LIN {X 0,Y 234.422,Z 1241.034,A -85,B 0,C 180,E1 12160.817,E2 12160.817} C_VEL
LIN {X 0,Y 234.7,Z 1243.569,A -85,B 0,C 180,E1 12156.114,E2 12156.114} C_VEL
LIN {X 0,Y 234.933,Z 1244.858,A -85,B 0,C 180,E1 12151.951,E2 12151.951} C_VEL
LIN {X 0,Y 234.862,Z 1245.105,A -85,B 0,C 180,E1 12147.56,E2 12147.56} C_VEL
LIN {X 0,Y 234.495,Z 1244.211,A -85,B 0,C 180,E1 12143.143,E2 12143.143} C_VEL
LIN {X 0,Y 234.238,Z 1241.662,A -85,B 0,C 180,E1 12137.833,E2 12137.833} C_VEL
LIN {X 0,Y 234.641,Z 1237.828,A -85,B 0,C 180,E1 12132.645,E2 12132.645} C_VEL
LIN {X 0,Y 235.984,Z 1232.823,A -85,B 0,C 180,E1 12127.584,E2 12127.584} C_VEL
LIN {X 0,Y 238.388,Z 1226.853,A -85,B 0,C 180,E1 12122.775,E2 12122.775} C_VEL
LIN {X 0,Y 241.931,Z 1219.741,A -85,B 0,C 180,E1 12118.061,E2 12118.061} C_VEL
LIN {X 0,Y 246.951,Z 1211.097,A -85,B 0,C 180,E1 12113.292,E2 12113.292} C_VEL
LIN {X 0,Y 255.037,Z 1198.442,A -85,B 0,C 180,E1 12107.598,E2 12107.598} C_VEL
LIN {X 0,Y 263.314,Z 1186.109,A -85,B 0,C 180,E1 12103.119,E2 12103.119} C_VEL
LIN {X 0,Y 271.68,Z 1173.895,A -85,B 0,C 180,E1 12099.387,E2 12099.387} C_VEL
LIN {X 0,Y 281.892,Z 1159.042,A -85,B 0,C 180,E1 12095.572,E2 12095.572} C_VEL
LIN {X 0,Y 294.354,Z 1140.405,A -85,B 0,C 180,E1 12091.689,E2 12091.689} C_VEL
LIN {X 0,Y 304.874,Z 1124.088,A -85,B 0,C 180,E1 12088.877,E2 12088.877} C_VEL
LIN {X 0,Y 315.79,Z 1106.483,A -85,B 0,C 180,E1 12086.314,E2 12086.314} C_VEL
LIN {X 0,Y 329.357,Z 1083.216,A -85,B 0,C 180,E1 12083.534,E2 12083.534} C_VEL
LIN {X 0,Y 339.871,Z 1063.804,A -85,B 0,C 180,E1 12081.62,E2 12081.62} C_VEL
LIN {X 0,Y 350.253,Z 1043.318,A -85,B 0,C 180,E1 12079.913,E2 12079.913} C_VEL
LIN {X 0,Y 362.426,Z 1017.02,A -85,B 0,C 180,E1 12078.118,E2 12078.118} C_VEL
LIN {X 0,Y 371.635,Z 994.992,A -85,B 0,C 180,E1 12076.892,E2 12076.892} C_VEL
LIN {X 0,Y 380.378,Z 971.962,A -85,B 0,C 180,E1 12075.829,E2 12075.829} C_VEL
LIN {X 0,Y 389.853,Z 943.44,A -85,B 0,C 180,E1 12074.781,E2 12074.781} C_VEL
LIN {X 0,Y 396.646,Z 919.703,A -85,B 0,C 180,E1 12074.096,E2 12074.096} C_VEL
LIN {X 0,Y 403.05,Z 892.634,A -85,B 0,C 180,E1 12073.424,E2 12073.424} C_VEL
LIN {X 0,Y 408.019,Z 864.078,A -85,B 0,C 180,E1 12072.829,E2 12072.829} C_VEL
LIN {X 0,Y 438.374,Z 631.58,A -85,B 0,C 180,E1 12068.871,E2 12068.871} C_VEL
LIN {X 0,Y 430.511,Z 617.928,A -85,B 0,C 180,E1 12065.23,E2 12065.23} C_VEL
LIN {X 0,Y 424.425,Z 607.912,A -85,B 0,C 180,E1 12062.059,E2 12062.059} C_VEL
LIN {X 0,Y 419.752,Z 600.312,A -85,B 0,C 180,E1 12059.318,E2 12059.318} C_VEL
LIN {X 0,Y 414.682,Z 592.173,A -85,B 0,C 180,E1 12055.99,E2 12055.99} C_VEL
LIN {X 0,Y 409.745,Z 584.609,A -85,B 0,C 180,E1 12052.287,E2 12052.287} C_VEL
LIN {X 0,Y 405.001,Z 577.41,A -85,B 0,C 180,E1 12048.031,E2 12048.031} C_VEL
LIN {X 0,Y 401.994,Z 572.607,A -85,B 0,C 180,E1 12044.713,E2 12044.713} C_VEL
LIN {X 0,Y 399.497,Z 568.951,A -85,B 0,C 180,E1 12041.466,E2 12041.466} C_VEL
LIN {X 0,Y 396.651,Z 566.18,A -85,B 0,C 180,E1 12036.939,E2 12036.939} C_VEL
LIN {X 0,Y 395.172,Z 563.252,A -85,B 0,C 180,E1 12033.274,E2 12033.274} C_VEL
LIN {X 0,Y 393.773,Z 562.552,A -85,B 0,C 180,E1 12028.839,E2 12028.839} C_VEL
LIN {X 0,Y 393.434,Z 562.231,A -85,B 0,C 180,E1 12024.165,E2 12024.165} C_VEL
LIN {X 0,Y 393.968,Z 562.553,A -85,B 0,C 180,E1 12019.363,E2 12019.363} C_VEL
LIN {X 0,Y 395.759,Z 563.395,A -85,B 0,C 180,E1 12014.617,E2 12014.617} C_VEL
LIN {X 0,Y 397.872,Z 567.235,A -85,B 0,C 180,E1 12010.183,E2 12010.183} C_VEL
LIN {X 0,Y 400.684,Z 569.721,A -85,B 0,C 180,E1 12006.53,E2 12006.53} C_VEL
LIN {X 0,Y 403.712,Z 573.853,A -85,B 0,C 180,E1 12003.16,E2 12003.16} C_VEL
LIN {X 0,Y 405.461,Z 575.63,A -85,B 0,C 180,E1 12001.603,E2 12001.603} C_VEL
LIN {X 0,Y 409.899,Z 581.322,A -85,B 0,C 180,E1 11997.927,E2 11997.927} C_VEL
LIN {X 0,Y 414.198,Z 586.829,A -85,B 0,C 180,E1 11994.906,E2 11994.906} C_VEL
LIN {X 0,Y 418.573,Z 592.702,A -85,B 0,C 180,E1 11992.174,E2 11992.174} C_VEL
LIN {X 0,Y 423.93,Z 599.787,A -85,B 0,C 180,E1 11989.245,E2 11989.245} C_VEL
LIN {X 0,Y 431.223,Z 610.33,A -85,B 0,C 180,E1 11985.706,E2 11985.706} C_VEL
LIN {X 0,Y 434.102,Z 614.761,A -85,B 0,C 180,E1 11984.42,E2 11984.42} C_VEL
LIN {X 0,Y 410.189,Z 798.407,A -85,B 0,C 180,E1 11981.329,E2 11981.329} C_VEL
LIN {X 0,Y 404.726,Z 829.257,A -85,B 0,C 180,E1 11980.609,E2 11980.609} C_VEL
LIN {X 0,Y 399.267,Z 853.642,A -85,B 0,C 180,E1 11979.878,E2 11979.878} C_VEL
LIN {X 0,Y 392.019,Z 880.927,A -85,B 0,C 180,E1 11978.876,E2 11978.876} C_VEL
LIN {X 0,Y 383.756,Z 906.782,A -85,B 0,C 180,E1 11977.701,E2 11977.701} C_VEL
LIN {X 0,Y 375.923,Z 928.552,A -85,B 0,C 180,E1 11976.525,E2 11976.525} C_VEL
LIN {X 0,Y 365.908,Z 953.393,A -85,B 0,C 180,E1 11974.938,E2 11974.938} C_VEL
LIN {X 0,Y 355.708,Z 975.722,A -85,B 0,C 180,E1 11973.223,E2 11973.223} C_VEL
LIN {X 0,Y 346.424,Z 994.396,A -85,B 0,C 180,E1 11971.551,E2 11971.551} C_VEL
LIN {X 0,Y 334.99,Z 1015.745,A -85,B 0,C 180,E1 11969.307,E2 11969.307} C_VEL
LIN {X 0,Y 323.122,Z 1035.835,A -85,B 0,C 180,E1 11966.747,E2 11966.747} C_VEL
LIN {X 0,Y 313.441,Z 1051.217,A -85,B 0,C 180,E1 11964.442,E2 11964.442} C_VEL
LIN {X 0,Y 303.132,Z 1066.743,A -85,B 0,C 180,E1 11961.716,E2 11961.716} C_VEL
LIN {X 0,Y 290.893,Z 1084.278,A -85,B 0,C 180,E1 11958.024,E2 11958.024} C_VEL
LIN {X 0,Y 280.853,Z 1097.923,A -85,B 0,C 180,E1 11954.514,E2 11954.514} C_VEL
LIN {X 0,Y 272.294,Z 1109.294,A -85,B 0,C 180,E1 11951.057,E2 11951.057} C_VEL
LIN {X 0,Y 264.585,Z 1119.425,A -85,B 0,C 180,E1 11947.433,E2 11947.433} C_VEL
LIN {X 0,Y 257.304,Z 1129.055,A -85,B 0,C 180,E1 11943.354,E2 11943.354} C_VEL
LIN {X 0,Y 249.783,Z 1139.381,A -85,B 0,C 180,E1 11938.065,E2 11938.065} C_VEL
LIN {X 0,Y 243.962,Z 1147.695,A -85,B 0,C 180,E1 11932.658,E2 11932.658} C_VEL
LIN {X 0,Y 240.175,Z 1153.774,A -85,B 0,C 180,E1 11927.821,E2 11927.821} C_VEL
LIN {X 0,Y 237.555,Z 1158.78,A -85,B 0,C 180,E1 11922.915,E2 11922.915} C_VEL
LIN {X 0,Y 235.895,Z 1162.839,A -85,B 0,C 180,E1 11917.924,E2 11917.924} C_VEL
LIN {X 0,Y 235.088,Z 1166.152,A -85,B 0,C 180,E1 11912.634,E2 11912.634} C_VEL
LIN {X 0,Y 234.883,Z 1168.717,A -85,B 0,C 180,E1 11906.823,E2 11906.823} C_VEL
LIN {X 0,Y 235.264,Z 1170.099,A -85,B 0,C 180,E1 11901.178,E2 11901.178} C_VEL
LIN {X 0,Y 236.121,Z 1170.572,A -85,B 0,C 180,E1 11895.977,E2 11895.977} C_VEL
LIN {X 0,Y 237.598,Z 1170.328,A -85,B 0,C 180,E1 11891.162,E2 11891.162} C_VEL
LIN {X 0,Y 240.343,Z 1169.243,A -85,B 0,C 180,E1 11885.97,E2 11885.97} C_VEL
LIN {X 0,Y 245.416,Z 1166.877,A -85,B 0,C 180,E1 11879.767,E2 11879.767} C_VEL
LIN {X 0,Y 253.48,Z 1162.729,A -85,B 0,C 180,E1 11873.204,E2 11873.204} C_VEL
LIN {X 0,Y 263.365,Z 1157.655,A -85,B 0,C 180,E1 11867.502,E2 11867.502} C_VEL
LIN {X 0,Y 278.43,Z 1149.865,A -85,B 0,C 180,E1 11861.143,E2 11861.143} C_VEL
LIN {X 0,Y 293.315,Z 1142.328,A -85,B 0,C 180,E1 11856.451,E2 11856.451} C_VEL
LIN {X 0,Y 295.573,Z 1141.406,A -85,B 0,C 180,E1 11855.547,E2 11855.547} C_VEL
LIN {X 0,Y 299.463,Z 1140.539,A -85,B 0,C 180,E1 11852.868,E2 11852.868} C_VEL
LIN {X 0,Y 301.764,Z 1139.659,A -85,B 0,C 180,E1 11852.154,E2 11852.154} C_VEL
LIN {X 0,Y 301.939,Z 1139.636,A -85,B 0,C 180,E1 11852.059,E2 11852.059} C_VEL
LIN {X 0,Y 275.793,Z 1163.771,A -85,B 0,C 180,E1 11845.384,E2 11845.384} C_VEL
LIN {X 0,Y 256.224,Z 1185.319,A -85,B 0,C 180,E1 11837.854,E2 11837.854} C_VEL
LIN {X 0,Y 245.979,Z 1198.298,A -85,B 0,C 180,E1 11832.284,E2 11832.284} C_VEL
LIN {X 0,Y 238.828,Z 1208.557,A -85,B 0,C 180,E1 11827.076,E2 11827.076} C_VEL
LIN {X 0,Y 233.731,Z 1217.045,A -85,B 0,C 180,E1 11822.036,E2 11822.036} C_VEL
LIN {X 0,Y 230.106,Z 1224.436,A -85,B 0,C 180,E1 11816.866,E2 11816.866} C_VEL
LIN {X 0,Y 227.883,Z 1230.405,A -85,B 0,C 180,E1 11811.898,E2 11811.898} C_VEL
LIN {X 0,Y 226.73,Z 1235.549,A -85,B 0,C 180,E1 11806.657,E2 11806.657} C_VEL
LIN {X 0,Y 226.486,Z 1239.507,A -85,B 0,C 180,E1 11801.452,E2 11801.452} C_VEL
LIN {X 0,Y 226.746,Z 1242.103,A -85,B 0,C 180,E1 11796.583,E2 11796.583} C_VEL
LIN {X 0,Y 227.037,Z 1243.443,A -85,B 0,C 180,E1 11792.271,E2 11792.271} C_VEL
LIN {X 0,Y 226.992,Z 1243.728,A -85,B 0,C 180,E1 11787.728,E2 11787.728} C_VEL
LIN {X 0,Y 226.604,Z 1242.842,A -85,B 0,C 180,E1 11783.128,E2 11783.128} C_VEL
LIN {X 0,Y 226.332,Z 1240.38,A -85,B 0,C 180,E1 11777.757,E2 11777.757} C_VEL
LIN {X 0,Y 226.769,Z 1236.476,A -85,B 0,C 180,E1 11772.288,E2 11772.288} C_VEL
LIN {X 0,Y 228.112,Z 1231.74,A -85,B 0,C 180,E1 11767.311,E2 11767.311} C_VEL
LIN {X 0,Y 230.597,Z 1225.838,A -85,B 0,C 180,E1 11762.357,E2 11762.357} C_VEL
LIN {X 0,Y 234.075,Z 1219.147,A -85,B 0,C 180,E1 11757.727,E2 11757.727} C_VEL
LIN {X 0,Y 238.931,Z 1211.085,A -85,B 0,C 180,E1 11753.064,E2 11753.064} C_VEL
LIN {X 0,Y 245.664,Z 1200.834,A -85,B 0,C 180,E1 11748.126,E2 11748.126} C_VEL
LIN {X 0,Y 255.633,Z 1186.526,A -85,B 0,C 180,E1 11742.585,E2 11742.585} C_VEL
LIN {X 0,Y 264.682,Z 1173.72,A -85,B 0,C 180,E1 11738.558,E2 11738.558} C_VEL
LIN {X 0,Y 273.854,Z 1160.76,A -85,B 0,C 180,E1 11735.13,E2 11735.13} C_VEL
LIN {X 0,Y 286.053,Z 1143.32,A -85,B 0,C 180,E1 11731.281,E2 11731.281} C_VEL
LIN {X 0,Y 298.71,Z 1124.262,A -85,B 0,C 180,E1 11727.909,E2 11727.909} C_VEL
LIN {X 0,Y 309.201,Z 1107.816,A -85,B 0,C 180,E1 11725.474,E2 11725.474} C_VEL
LIN {X 0,Y 321.711,Z 1087.238,A -85,B 0,C 180,E1 11722.918,E2 11722.918} C_VEL
LIN {X 0,Y 334.128,Z 1065.005,A -85,B 0,C 180,E1 11720.678,E2 11720.678} C_VEL
LIN {X 0,Y 344.265,Z 1045.498,A -85,B 0,C 180,E1 11719.037,E2 11719.037} C_VEL
LIN {X 0,Y 355.267,Z 1022.699,A -85,B 0,C 180,E1 11717.428,E2 11717.428} C_VEL
LIN {X 0,Y 366.125,Z 997.612,A -85,B 0,C 180,E1 11715.992,E2 11715.992} C_VEL
LIN {X 0,Y 374.666,Z 975.771,A -85,B 0,C 180,E1 11714.967,E2 11714.967} C_VEL
LIN {X 0,Y 383.02,Z 952.046,A -85,B 0,C 180,E1 11714.051,E2 11714.051} C_VEL
LIN {X 0,Y 391.563,Z 923.901,A -85,B 0,C 180,E1 11713.195,E2 11713.195} C_VEL
LIN {X 0,Y 397.58,Z 899.939,A -85,B 0,C 180,E1 11712.594,E2 11712.594} C_VEL
LIN {X 0,Y 402.75,Z 874.159,A -85,B 0,C 180,E1 11712.021,E2 11712.021} C_VEL
LIN {X 0,Y 408.292,Z 835.423,A -85,B 0,C 180,E1 11711.309,E2 11711.309} C_VEL
LIN {X 0,Y 434.7,Z 636.533,A -85,B 0,C 180,E1 11707.966,E2 11707.966} C_VEL
LIN {X 0,Y 427.973,Z 624.737,A -85,B 0,C 180,E1 11704.758,E2 11704.758} C_VEL
LIN {X 0,Y 422.268,Z 615.214,A -85,B 0,C 180,E1 11701.727,E2 11701.727} C_VEL
LIN {X 0,Y 417.624,Z 607.612,A -85,B 0,C 180,E1 11698.971,E2 11698.971} C_VEL
LIN {X 0,Y 412.699,Z 599.634,A -85,B 0,C 180,E1 11695.693,E2 11695.693} C_VEL
LIN {X 0,Y 408.17,Z 592.622,A -85,B 0,C 180,E1 11692.257,E2 11692.257} C_VEL
LIN {X 0,Y 403.583,Z 585.486,A -85,B 0,C 180,E1 11688.129,E2 11688.129} C_VEL
LIN {X 0,Y 400.287,Z 580.297,A -85,B 0,C 180,E1 11684.497,E2 11684.497} C_VEL
LIN {X 0,Y 397.874,Z 576.75,A -85,B 0,C 180,E1 11681.337,E2 11681.337} C_VEL
LIN {X 0,Y 394.986,Z 573.915,A -85,B 0,C 180,E1 11676.74,E2 11676.74} C_VEL
LIN {X 0,Y 393.634,Z 571.113,A -85,B 0,C 180,E1 11673.281,E2 11673.281} C_VEL
LIN {X 0,Y 392.232,Z 570.402,A -85,B 0,C 180,E1 11668.835,E2 11668.835} C_VEL
LIN {X 0,Y 391.893,Z 570.084,A -85,B 0,C 180,E1 11664.228,E2 11664.228} C_VEL
LIN {X 0,Y 392.428,Z 570.401,A -85,B 0,C 180,E1 11659.401,E2 11659.401} C_VEL
LIN {X 0,Y 394.169,Z 571.209,A -85,B 0,C 180,E1 11654.742,E2 11654.742} C_VEL
LIN {X 0,Y 396.379,Z 575.142,A -85,B 0,C 180,E1 11650.152,E2 11650.152} C_VEL
LIN {X 0,Y 399.044,Z 577.472,A -85,B 0,C 180,E1 11646.694,E2 11646.694} C_VEL
LIN {X 0,Y 402.228,Z 581.766,A -85,B 0,C 180,E1 11643.154,E2 11643.154} C_VEL
LIN {X 0,Y 403.777,Z 583.406,A -85,B 0,C 180,E1 11641.75,E2 11641.75} C_VEL
LIN {X 0,Y 408.145,Z 589.012,A -85,B 0,C 180,E1 11638.122,E2 11638.122} C_VEL
LIN {X 0,Y 412.383,Z 594.497,A -85,B 0,C 180,E1 11635.107,E2 11635.107} C_VEL
LIN {X 0,Y 416.581,Z 600.152,A -85,B 0,C 180,E1 11632.468,E2 11632.468} C_VEL
LIN {X 0,Y 421.918,Z 607.271,A -85,B 0,C 180,E1 11629.521,E2 11629.521} C_VEL
LIN {X 0,Y 429.179,Z 617.87,A -85,B 0,C 180,E1 11625.957,E2 11625.957} C_VEL
LIN {X 0,Y 430.532,Z 620.121,A -85,B 0,C 180,E1 11625.326,E2 11625.326} C_VEL
LIN {X 0,Y 406.793,Z 798.694,A -85,B 0,C 180,E1 11622.345,E2 11622.345} C_VEL
LIN {X 0,Y 401.234,Z 829.703,A -85,B 0,C 180,E1 11621.631,E2 11621.631} C_VEL
LIN {X 0,Y 395.799,Z 853.696,A -85,B 0,C 180,E1 11620.922,E2 11620.922} C_VEL
LIN {X 0,Y 388.651,Z 880.41,A -85,B 0,C 180,E1 11619.96,E2 11619.96} C_VEL
LIN {X 0,Y 380.1,Z 906.91,A -85,B 0,C 180,E1 11618.776,E2 11618.776} C_VEL
LIN {X 0,Y 372.259,Z 928.403,A -85,B 0,C 180,E1 11617.631,E2 11617.631} C_VEL
LIN {X 0,Y 362.311,Z 952.866,A -85,B 0,C 180,E1 11616.098,E2 11616.098} C_VEL
LIN {X 0,Y 351.313,Z 976.538,A -85,B 0,C 180,E1 11614.3,E2 11614.3} C_VEL
LIN {X 0,Y 342.082,Z 994.772,A -85,B 0,C 180,E1 11612.681,E2 11612.681} C_VEL
LIN {X 0,Y 330.982,Z 1015.11,A -85,B 0,C 180,E1 11610.567,E2 11610.567} C_VEL
LIN {X 0,Y 318.185,Z 1036.478,A -85,B 0,C 180,E1 11607.877,E2 11607.877} C_VEL
LIN {X 0,Y 307.923,Z 1052.44,A -85,B 0,C 180,E1 11605.486,E2 11605.486} C_VEL
LIN {X 0,Y 297.791,Z 1067.386,A -85,B 0,C 180,E1 11602.864,E2 11602.864} C_VEL
LIN {X 0,Y 285.709,Z 1084.402,A -85,B 0,C 180,E1 11599.311,E2 11599.311} C_VEL
LIN {X 0,Y 274.386,Z 1099.39,A -85,B 0,C 180,E1 11595.437,E2 11595.437} C_VEL
LIN {X 0,Y 265.188,Z 1111.244,A -85,B 0,C 180,E1 11591.763,E2 11591.763} C_VEL
LIN {X 0,Y 256.212,Z 1122.705,A -85,B 0,C 180,E1 11587.515,E2 11587.515} C_VEL
LIN {X 0,Y 246.831,Z 1134.724,A -85,B 0,C 180,E1 11581.972,E2 11581.972} C_VEL
LIN {X 0,Y 240.673,Z 1142.891,A -85,B 0,C 180,E1 11577.311,E2 11577.311} C_VEL
LIN {X 0,Y 235.936,Z 1149.613,A -85,B 0,C 180,E1 11572.698,E2 11572.698} C_VEL
LIN {X 0,Y 232.166,Z 1155.527,A -85,B 0,C 180,E1 11567.79,E2 11567.79} C_VEL
LIN {X 0,Y 229.434,Z 1160.696,A -85,B 0,C 180,E1 11562.493,E2 11562.493} C_VEL
LIN {X 0,Y 227.574,Z 1165.693,A -85,B 0,C 180,E1 11555.758,E2 11555.758} C_VEL
LIN {X 0,Y 227.033,Z 1168.637,A -85,B 0,C 180,E1 11550.138,E2 11550.138} C_VEL
LIN {X 0,Y 227.051,Z 1170.514,A -85,B 0,C 180,E1 11545.01,E2 11545.01} C_VEL
LIN {X 0,Y 227.501,Z 1171.634,A -85,B 0,C 180,E1 11540.049,E2 11540.049} C_VEL
LIN {X 0,Y 228.425,Z 1172.094,A -85,B 0,C 180,E1 11535.227,E2 11535.227} C_VEL
LIN {X 0,Y 230.104,Z 1171.893,A -85,B 0,C 180,E1 11530.263,E2 11530.263} C_VEL
LIN {X 0,Y 233.156,Z 1170.882,A -85,B 0,C 180,E1 11524.92,E2 11524.92} C_VEL
LIN {X 0,Y 239.244,Z 1168.447,A -85,B 0,C 180,E1 11518.084,E2 11518.084} C_VEL
LIN {X 0,Y 248.147,Z 1164.309,A -85,B 0,C 180,E1 11511.426,E2 11511.426} C_VEL
LIN {X 0,Y 260.72,Z 1158.606,A -85,B 0,C 180,E1 11504.883,E2 11504.883} C_VEL
LIN {X 0,Y 279.21,Z 1149.934,A -85,B 0,C 180,E1 11498.048,E2 11498.048} C_VEL
LIN {X 0,Y 301.113,Z 1139.941,A -85,B 0,C 180,E1 11492.297,E2 11492.297} C_VEL
LIN {X 0,Y 301.764,Z 1139.659,A -85,B 0,C 180,E1 11492.154,E2 11492.154} C_VEL
LIN {X 0,Y 302.162,Z 1139.777,A -85,B 0,C 180,E1 11491.778,E2 11491.778} C_VEL
LIN {X 0,Y 300.773,Z 1141.241,A -85,B 0,C 180,E1 11491.224,E2 11491.224} C_VEL
LIN {X 0,Y 296.315,Z 1144.749,A -85,B 0,C 180,E1 11490.576,E2 11490.576} C_VEL
LIN {X 0,Y 282.499,Z 1154.252,A -85,B 0,C 180,E1 11489.503,E2 11489.503} C_VEL
LIN {X 0,Y 278.089,Z 1157.541,A -85,B 0,C 180,E1 11488.81,E2 11488.81} C_VEL
LIN {X 0,Y 277.288,Z 1158.24,A -85,B 0,C 180,E1 11488.611,E2 11488.611} C_VEL
LIN {X 0,Y 253.039,Z 1182.018,A -85,B 0,C 180,E1 11480.402,E2 11480.402} C_VEL
LIN {X 0,Y 240.686,Z 1196.16,A -85,B 0,C 180,E1 11474.26,E2 11474.26} C_VEL
LIN {X 0,Y 232.339,Z 1207.025,A -85,B 0,C 180,E1 11468.609,E2 11468.609} C_VEL
LIN {X 0,Y 226.553,Z 1215.843,A -85,B 0,C 180,E1 11463.179,E2 11463.179} C_VEL
LIN {X 0,Y 222.525,Z 1223.309,A -85,B 0,C 180,E1 11457.724,E2 11457.724} C_VEL
LIN {X 0,Y 220.065,Z 1229.357,A -85,B 0,C 180,E1 11452.436,E2 11452.436} C_VEL
LIN {X 0,Y 218.853,Z 1234.201,A -85,B 0,C 180,E1 11447.275,E2 11447.275} C_VEL
LIN {X 0,Y 218.54,Z 1237.967,A -85,B 0,C 180,E1 11442.149,E2 11442.149} C_VEL
LIN {X 0,Y 218.771,Z 1240.528,A -85,B 0,C 180,E1 11437.342,E2 11437.342} C_VEL
LIN {X 0,Y 219.117,Z 1241.981,A -85,B 0,C 180,E1 11432.877,E2 11432.877} C_VEL
LIN {X 0,Y 219.13,Z 1242.384,A -85,B 0,C 180,E1 11428.17,E2 11428.17} C_VEL
LIN {X 0,Y 218.743,Z 1241.599,A -85,B 0,C 180,E1 11423.438,E2 11423.438} C_VEL
LIN {X 0,Y 218.426,Z 1239.193,A -85,B 0,C 180,E1 11417.844,E2 11417.844} C_VEL
LIN {X 0,Y 218.852,Z 1235.35,A -85,B 0,C 180,E1 11412.175,E2 11412.175} C_VEL
LIN {X 0,Y 220.356,Z 1230.382,A -85,B 0,C 180,E1 11406.749,E2 11406.749} C_VEL
LIN {X 0,Y 223.001,Z 1224.465,A -85,B 0,C 180,E1 11401.623,E2 11401.623} C_VEL
LIN {X 0,Y 226.702,Z 1217.743,A -85,B 0,C 180,E1 11396.845,E2 11396.845} C_VEL
LIN {X 0,Y 231.95,Z 1209.439,A -85,B 0,C 180,E1 11391.944,E2 11391.944} C_VEL
LIN {X 0,Y 240.114,Z 1197.738,A -85,B 0,C 180,E1 11386.271,E2 11386.271} C_VEL
LIN {X 0,Y 249.719,Z 1184.4,A -85,B 0,C 180,E1 11381.17,E2 11381.17} C_VEL
LIN {X 0,Y 258.803,Z 1172.049,A -85,B 0,C 180,E1 11377.262,E2 11377.262} C_VEL
LIN {X 0,Y 269.514,Z 1157.448,A -85,B 0,C 180,E1 11373.412,E2 11373.412} C_VEL
LIN {X 0,Y 282.806,Z 1138.8,A -85,B 0,C 180,E1 11369.436,E2 11369.436} C_VEL
LIN {X 0,Y 293.673,Z 1122.857,A -85,B 0,C 180,E1 11366.653,E2 11366.653} C_VEL
LIN {X 0,Y 304.682,Z 1105.965,A -85,B 0,C 180,E1 11364.173,E2 11364.173} C_VEL
LIN {X 0,Y 318.14,Z 1084.13,A -85,B 0,C 180,E1 11361.52,E2 11361.52} C_VEL
LIN {X 0,Y 330.237,Z 1062.753,A -85,B 0,C 180,E1 11359.413,E2 11359.413} C_VEL
LIN {X 0,Y 340.729,Z 1042.858,A -85,B 0,C 180,E1 11357.77,E2 11357.77} C_VEL
LIN {X 0,Y 352.76,Z 1018.101,A -85,B 0,C 180,E1 11356.081,E2 11356.081} C_VEL
LIN {X 0,Y 362.978,Z 994.576,A -85,B 0,C 180,E1 11354.787,E2 11354.787} C_VEL
LIN {X 0,Y 371.662,Z 972.557,A -85,B 0,C 180,E1 11353.786,E2 11353.786} C_VEL
LIN {X 0,Y 381.161,Z 945.476,A -85,B 0,C 180,E1 11352.79,E2 11352.79} C_VEL
LIN {X 0,Y 388.711,Z 920.179,A -85,B 0,C 180,E1 11352.07,E2 11352.07} C_VEL
LIN {X 0,Y 394.526,Z 896.939,A -85,B 0,C 180,E1 11351.499,E2 11351.499} C_VEL
LIN {X 0,Y 400.202,Z 868.074,A -85,B 0,C 180,E1 11350.876,E2 11350.876} C_VEL
LIN {X 0,Y 407.304,Z 816.655,A -85,B 0,C 180,E1 11349.97,E2 11349.97} C_VEL
LIN {X 0,Y 431.165,Z 641.595,A -85,B 0,C 180,E1 11347.06,E2 11347.06} C_VEL
LIN {X 0,Y 424.708,Z 630.234,A -85,B 0,C 180,E1 11343.881,E2 11343.881} C_VEL
LIN {X 0,Y 418.475,Z 619.575,A -85,B 0,C 180,E1 11340.411,E2 11340.411} C_VEL
LIN {X 0,Y 412.079,Z 609.24,A -85,B 0,C 180,E1 11336.313,E2 11336.313} C_VEL
LIN {X 0,Y 407.153,Z 601.482,A -85,B 0,C 180,E1 11332.663,E2 11332.663} C_VEL
LIN {X 0,Y 404.391,Z 597.255,A -85,B 0,C 180,E1 11330.32,E2 11330.32} C_VEL
LIN {X 0,Y 401.42,Z 592.59,A -85,B 0,C 180,E1 11327.484,E2 11327.484} C_VEL
LIN {X 0,Y 398.585,Z 587.986,A -85,B 0,C 180,E1 11324.28,E2 11324.28} C_VEL
LIN {X 0,Y 396.333,Z 584.602,A -85,B 0,C 180,E1 11321.313,E2 11321.313} C_VEL
LIN {X 0,Y 393.384,Z 581.722,A -85,B 0,C 180,E1 11316.639,E2 11316.639} C_VEL
LIN {X 0,Y 392.04,Z 578.925,A -85,B 0,C 180,E1 11313.164,E2 11313.164} C_VEL
LIN {X 0,Y 390.7,Z 578.255,A -85,B 0,C 180,E1 11308.871,E2 11308.871} C_VEL
LIN {X 0,Y 390.35,Z 577.935,A -85,B 0,C 180,E1 11304.265,E2 11304.265} C_VEL
LIN {X 0,Y 390.888,Z 578.249,A -85,B 0,C 180,E1 11299.439,E2 11299.439} C_VEL
LIN {X 0,Y 392.593,Z 579.04,A -85,B 0,C 180,E1 11294.821,E2 11294.821} C_VEL
LIN {X 0,Y 394.759,Z 582.904,A -85,B 0,C 180,E1 11290.323,E2 11290.323} C_VEL
LIN {X 0,Y 397.407,Z 585.224,A -85,B 0,C 180,E1 11286.86,E2 11286.86} C_VEL
LIN {X 0,Y 400.619,Z 589.562,A -85,B 0,C 180,E1 11283.267,E2 11283.267} C_VEL
LIN {X 0,Y 402.096,Z 591.18,A -85,B 0,C 180,E1 11281.898,E2 11281.898} C_VEL
LIN {X 0,Y 406.324,Z 596.624,A -85,B 0,C 180,E1 11278.355,E2 11278.355} C_VEL
LIN {X 0,Y 410.643,Z 602.266,A -85,B 0,C 180,E1 11275.263,E2 11275.263} C_VEL
LIN {X 0,Y 414.721,Z 607.772,A -85,B 0,C 180,E1 11272.691,E2 11272.691} C_VEL
LIN {X 0,Y 419.978,Z 614.868,A -85,B 0,C 180,E1 11269.759,E2 11269.759} C_VEL
LIN {X 0,Y 427.04,Z 625.276,A -85,B 0,C 180,E1 11266.248,E2 11266.248} C_VEL
LIN {X 0,Y 403.207,Z 800.417,A -85,B 0,C 180,E1 11263.343,E2 11263.343} C_VEL
LIN {X 0,Y 397.539,Z 831.173,A -85,B 0,C 180,E1 11262.636,E2 11262.636} C_VEL
LIN {X 0,Y 391.957,Z 855.307,A -85,B 0,C 180,E1 11261.925,E2 11261.925} C_VEL
LIN {X 0,Y 384.476,Z 882.596,A -85,B 0,C 180,E1 11260.944,E2 11260.944} C_VEL
LIN {X 0,Y 375.996,Z 908.327,A -85,B 0,C 180,E1 11259.799,E2 11259.799} C_VEL
LIN {X 0,Y 367.899,Z 930.148,A -85,B 0,C 180,E1 11258.644,E2 11258.644} C_VEL
LIN {X 0,Y 357.452,Z 955.255,A -85,B 0,C 180,E1 11257.07,E2 11257.07} C_VEL
LIN {X 0,Y 346.783,Z 977.834,A -85,B 0,C 180,E1 11255.362,E2 11255.362} C_VEL
LIN {X 0,Y 336.878,Z 997.036,A -85,B 0,C 180,E1 11253.659,E2 11253.659} C_VEL
LIN {X 0,Y 324.315,Z 1019.4,A -85,B 0,C 180,E1 11251.297,E2 11251.297} C_VEL
LIN {X 0,Y 312.728,Z 1038.135,A -85,B 0,C 180,E1 11248.901,E2 11248.901} C_VEL
LIN {X 0,Y 302.511,Z 1053.657,A -85,B 0,C 180,E1 11246.569,E2 11246.569} C_VEL
LIN {X 0,Y 292.022,Z 1068.759,A -85,B 0,C 180,E1 11243.907,E2 11243.907} C_VEL
LIN {X 0,Y 279.613,Z 1085.757,A -85,B 0,C 180,E1 11240.325,E2 11240.325} C_VEL
LIN {X 0,Y 268.342,Z 1100.276,A -85,B 0,C 180,E1 11236.542,E2 11236.542} C_VEL
LIN {X 0,Y 259.145,Z 1111.819,A -85,B 0,C 180,E1 11232.948,E2 11232.948} C_VEL
LIN {X 0,Y 250.579,Z 1122.413,A -85,B 0,C 180,E1 11229.025,E2 11229.025} C_VEL
LIN {X 0,Y 241.298,Z 1134.052,A -85,B 0,C 180,E1 11223.803,E2 11223.803} C_VEL
LIN {X 0,Y 233.349,Z 1144.081,A -85,B 0,C 180,E1 11218.041,E2 11218.041} C_VEL
LIN {X 0,Y 228.243,Z 1151.066,A -85,B 0,C 180,E1 11213.119,E2 11213.119} C_VEL
LIN {X 0,Y 224.164,Z 1157.28,A -85,B 0,C 180,E1 11207.77,E2 11207.77} C_VEL
LIN {X 0,Y 221.065,Z 1163.226,A -85,B 0,C 180,E1 11201.328,E2 11201.328} C_VEL
LIN {X 0,Y 219.579,Z 1167.268,A -85,B 0,C 180,E1 11195.332,E2 11195.332} C_VEL
LIN {X 0,Y 219.133,Z 1169.926,A -85,B 0,C 180,E1 11190.128,E2 11190.128} C_VEL
LIN {X 0,Y 219.168,Z 1171.888,A -85,B 0,C 180,E1 11184.788,E2 11184.788} C_VEL
LIN {X 0,Y 219.685,Z 1173.097,A -85,B 0,C 180,E1 11179.586,E2 11179.586} C_VEL
LIN {X 0,Y 220.767,Z 1173.62,A -85,B 0,C 180,E1 11174.425,E2 11174.425} C_VEL
LIN {X 0,Y 222.814,Z 1173.456,A -85,B 0,C 180,E1 11169.037,E2 11169.037} C_VEL
LIN {X 0,Y 226.363,Z 1172.464,A -85,B 0,C 180,E1 11163.37,E2 11163.37} C_VEL
LIN {X 0,Y 233.502,Z 1169.924,A -85,B 0,C 180,E1 11156.132,E2 11156.132} C_VEL
LIN {X 0,Y 243.502,Z 1165.818,A -85,B 0,C 180,E1 11149.351,E2 11149.351} C_VEL
LIN {X 0,Y 257.818,Z 1159.904,A -85,B 0,C 180,E1 11142.562,E2 11142.562} C_VEL
LIN {X 0,Y 277.458,Z 1151.727,A -85,B 0,C 180,E1 11135.969,E2 11135.969} C_VEL
LIN {X 0,Y 292.187,Z 1145.694,A -85,B 0,C 180,E1 11132.186,E2 11132.186} C_VEL
LIN {X 0,Y 277.288,Z 1158.24,A -85,B 0,C 180,E1 11128.611,E2 11128.611} C_VEL
LIN {X 0,Y 272.552,Z 1162.19,A -85,B 0,C 180,E1 11127.615,E2 11127.615} C_VEL
LIN {X 0,Y 257.615,Z 1172.667,A -85,B 0,C 180,E1 11125.281,E2 11125.281} C_VEL
LIN {X 0,Y 253.807,Z 1175.745,A -85,B 0,C 180,E1 11124.273,E2 11124.273} C_VEL
LIN {X 0,Y 236.34,Z 1193.39,A -85,B 0,C 180,E1 11116.691,E2 11116.691} C_VEL
LIN {X 0,Y 226.399,Z 1205.124,A -85,B 0,C 180,E1 11110.482,E2 11110.482} C_VEL
LIN {X 0,Y 219.21,Z 1215.079,A -85,B 0,C 180,E1 11104.127,E2 11104.127} C_VEL
LIN {X 0,Y 213.708,Z 1224.89,A -85,B 0,C 180,E1 11096.39,E2 11096.39} C_VEL
LIN {X 0,Y 211.221,Z 1231.706,A -85,B 0,C 180,E1 11089.352,E2 11089.352} C_VEL
LIN {X 0,Y 210.59,Z 1235.932,A -85,B 0,C 180,E1 11083.733,E2 11083.733} C_VEL
LIN {X 0,Y 210.761,Z 1238.824,A -85,B 0,C 180,E1 11078.457,E2 11078.457} C_VEL
LIN {X 0,Y 211.192,Z 1240.509,A -85,B 0,C 180,E1 11073.529,E2 11073.529} C_VEL
LIN {X 0,Y 211.255,Z 1241.028,A -85,B 0,C 180,E1 11068.915,E2 11068.915} C_VEL
LIN {X 0,Y 210.959,Z 1240.403,A -85,B 0,C 180,E1 11064.288,E2 11064.288} C_VEL
LIN {X 0,Y 210.533,Z 1238.308,A -85,B 0,C 180,E1 11058.494,E2 11058.494} C_VEL
LIN {X 0,Y 210.94,Z 1234.194,A -85,B 0,C 180,E1 11052.055,E2 11052.055} C_VEL
LIN {X 0,Y 212.504,Z 1229.264,A -85,B 0,C 180,E1 11046.425,E2 11046.425} C_VEL
LIN {X 0,Y 215.264,Z 1223.37,A -85,B 0,C 180,E1 11041.114,E2 11041.114} C_VEL
LIN {X 0,Y 219.177,Z 1216.606,A -85,B 0,C 180,E1 11036.129,E2 11036.129} C_VEL
LIN {X 0,Y 224.501,Z 1208.557,A -85,B 0,C 180,E1 11031.208,E2 11031.208} C_VEL
LIN {X 0,Y 231.891,Z 1198.313,A -85,B 0,C 180,E1 11026.036,E2 11026.036} C_VEL
LIN {X 0,Y 242.606,Z 1184.091,A -85,B 0,C 180,E1 11020.318,E2 11020.318} C_VEL
LIN {X 0,Y 251.957,Z 1171.823,A -85,B 0,C 180,E1 11016.332,E2 11016.332} C_VEL
LIN {X 0,Y 261.75,Z 1158.862,A -85,B 0,C 180,E1 11012.818,E2 11012.818} C_VEL
LIN {X 0,Y 273.718,Z 1142.73,A -85,B 0,C 180,E1 11009.185,E2 11009.185} C_VEL
LIN {X 0,Y 287.358,Z 1123.384,A -85,B 0,C 180,E1 11005.683,E2 11005.683} C_VEL
LIN {X 0,Y 298.587,Z 1106.638,A -85,B 0,C 180,E1 11003.188,E2 11003.188} C_VEL
LIN {X 0,Y 310.733,Z 1087.539,A -85,B 0,C 180,E1 11000.809,E2 11000.809} C_VEL
LIN {X 0,Y 324.596,Z 1063.941,A -85,B 0,C 180,E1 10998.422,E2 10998.422} C_VEL
LIN {X 0,Y 335.244,Z 1044.278,A -85,B 0,C 180,E1 10996.786,E2 10996.786} C_VEL
LIN {X 0,Y 346.182,Z 1022.497,A -85,B 0,C 180,E1 10995.271,E2 10995.271} C_VEL
LIN {X 0,Y 358.248,Z 995.74,A -85,B 0,C 180,E1 10993.767,E2 10993.767} C_VEL
LIN {X 0,Y 367.043,Z 973.97,A -85,B 0,C 180,E1 10992.777,E2 10992.777} C_VEL
LIN {X 0,Y 375.98,Z 949.329,A -85,B 0,C 180,E1 10991.86,E2 10991.86} C_VEL
LIN {X 0,Y 384.819,Z 920.801,A -85,B 0,C 180,E1 10991.036,E2 10991.036} C_VEL
LIN {X 0,Y 390.941,Z 896.874,A -85,B 0,C 180,E1 10990.454,E2 10990.454} C_VEL
LIN {X 0,Y 396.731,Z 868.302,A -85,B 0,C 180,E1 10989.84,E2 10989.84} C_VEL
LIN {X 0,Y 404.892,Z 810.837,A -85,B 0,C 180,E1 10988.835,E2 10988.835} C_VEL
LIN {X 0,Y 427.68,Z 646.546,A -85,B 0,C 180,E1 10986.128,E2 10986.128} C_VEL
LIN {X 0,Y 420.731,Z 634.384,A -85,B 0,C 180,E1 10982.588,E2 10982.588} C_VEL
LIN {X 0,Y 414.623,Z 624.067,A -85,B 0,C 180,E1 10979.033,E2 10979.033} C_VEL
LIN {X 0,Y 409.051,Z 614.975,A -85,B 0,C 180,E1 10975.303,E2 10975.303} C_VEL
LIN {X 0,Y 404.83,Z 608.356,A -85,B 0,C 180,E1 10972.05,E2 10972.05} C_VEL
LIN {X 0,Y 402.068,Z 604.104,A -85,B 0,C 180,E1 10969.613,E2 10969.613} C_VEL
LIN {X 0,Y 399.643,Z 600.178,A -85,B 0,C 180,E1 10967.207,E2 10967.207} C_VEL
LIN {X 0,Y 396.889,Z 595.675,A -85,B 0,C 180,E1 10964.061,E2 10964.061} C_VEL
LIN {X 0,Y 394.636,Z 592.347,A -85,B 0,C 180,E1 10961.076,E2 10961.076} C_VEL
LIN {X 0,Y 391.693,Z 589.409,A -85,B 0,C 180,E1 10956.373,E2 10956.373} C_VEL
LIN {X 0,Y 390.438,Z 586.73,A -85,B 0,C 180,E1 10953.024,E2 10953.024} C_VEL
LIN {X 0,Y 389.133,Z 586.094,A -85,B 0,C 180,E1 10948.732,E2 10948.732} C_VEL
LIN {X 0,Y 388.806,Z 585.773,A -85,B 0,C 180,E1 10943.919,E2 10943.919} C_VEL
LIN {X 0,Y 389.39,Z 586.124,A -85,B 0,C 180,E1 10939.244,E2 10939.244} C_VEL
LIN {X 0,Y 391.045,Z 586.99,A -85,B 0,C 180,E1 10934.801,E2 10934.801} C_VEL
LIN {X 0,Y 393.304,Z 590.859,A -85,B 0,C 180,E1 10930.22,E2 10930.22} C_VEL
LIN {X 0,Y 395.82,Z 593.076,A -85,B 0,C 180,E1 10926.956,E2 10926.956} C_VEL
LIN {X 0,Y 399.183,Z 597.517,A -85,B 0,C 180,E1 10923.215,E2 10923.215} C_VEL
LIN {X 0,Y 400.419,Z 598.953,A -85,B 0,C 180,E1 10922.048,E2 10922.048} C_VEL
LIN {X 0,Y 404.646,Z 604.441,A -85,B 0,C 180,E1 10918.483,E2 10918.483} C_VEL
LIN {X 0,Y 408.68,Z 609.703,A -85,B 0,C 180,E1 10915.576,E2 10915.576} C_VEL
LIN {X 0,Y 413.078,Z 615.685,A -85,B 0,C 180,E1 10912.786,E2 10912.786} C_VEL
LIN {X 0,Y 418.223,Z 622.795,A -85,B 0,C 180,E1 10909.882,E2 10909.882} C_VEL
LIN {X 0,Y 423.535,Z 630.753,A -85,B 0,C 180,E1 10907.175,E2 10907.175} C_VEL
LIN {X 0,Y 399.897,Z 801.083,A -85,B 0,C 180,E1 10904.378,E2 10904.378} C_VEL
LIN {X 0,Y 394.095,Z 832.069,A -85,B 0,C 180,E1 10903.674,E2 10903.674} C_VEL
LIN {X 0,Y 388.412,Z 856.192,A -85,B 0,C 180,E1 10902.97,E2 10902.97} C_VEL
LIN {X 0,Y 381.011,Z 882.822,A -85,B 0,C 180,E1 10902.026,E2 10902.026} C_VEL
LIN {X 0,Y 372.284,Z 908.942,A -85,B 0,C 180,E1 10900.881,E2 10900.881} C_VEL
LIN {X 0,Y 363.786,Z 931.451,A -85,B 0,C 180,E1 10899.702,E2 10899.702} C_VEL
LIN {X 0,Y 353.141,Z 956.526,A -85,B 0,C 180,E1 10898.139,E2 10898.139} C_VEL
LIN {X 0,Y 342.828,Z 978.001,A -85,B 0,C 180,E1 10896.531,E2 10896.531} C_VEL
LIN {X 0,Y 333.196,Z 996.409,A -85,B 0,C 180,E1 10894.926,E2 10894.926} C_VEL
LIN {X 0,Y 322.402,Z 1015.509,A -85,B 0,C 180,E1 10892.979,E2 10892.979} C_VEL
LIN {X 0,Y 308.972,Z 1037.289,A -85,B 0,C 180,E1 10890.304,E2 10890.304} C_VEL
LIN {X 0,Y 297.773,Z 1054.041,A -85,B 0,C 180,E1 10887.823,E2 10887.823} C_VEL
LIN {X 0,Y 286.993,Z 1069.252,A -85,B 0,C 180,E1 10885.161,E2 10885.161} C_VEL
LIN {X 0,Y 273.984,Z 1086.652,A -85,B 0,C 180,E1 10881.497,E2 10881.497} C_VEL
LIN {X 0,Y 262.1,Z 1101.539,A -85,B 0,C 180,E1 10877.588,E2 10877.588} C_VEL
LIN {X 0,Y 252.762,Z 1112.92,A -85,B 0,C 180,E1 10874.004,E2 10874.004} C_VEL
LIN {X 0,Y 244.127,Z 1123.269,A -85,B 0,C 180,E1 10870.127,E2 10870.127} C_VEL
LIN {X 0,Y 234.874,Z 1134.449,A -85,B 0,C 180,E1 10865.064,E2 10865.064} C_VEL
LIN {X 0,Y 226.527,Z 1144.628,A -85,B 0,C 180,E1 10859.202,E2 10859.202} C_VEL
LIN {X 0,Y 221.018,Z 1151.819,A -85,B 0,C 180,E1 10854.077,E2 10854.077} C_VEL
LIN {X 0,Y 217.017,Z 1157.595,A -85,B 0,C 180,E1 10849.08,E2 10849.08} C_VEL
LIN {X 0,Y 214.226,Z 1162.364,A -85,B 0,C 180,E1 10844.047,E2 10844.047} C_VEL
LIN {X 0,Y 212.315,Z 1166.543,A -85,B 0,C 180,E1 10838.578,E2 10838.578} C_VEL
LIN {X 0,Y 211.434,Z 1169.762,A -85,B 0,C 180,E1 10833.172,E2 10833.172} C_VEL
LIN {X 0,Y 211.167,Z 1172.239,A -85,B 0,C 180,E1 10827.648,E2 10827.648} C_VEL
LIN {X 0,Y 211.531,Z 1174.115,A -85,B 0,C 180,E1 10821.636,E2 10821.636} C_VEL
LIN {X 0,Y 212.745,Z 1175.133,A -85,B 0,C 180,E1 10814.981,E2 10814.981} C_VEL
LIN {X 0,Y 215.174,Z 1175.126,A -85,B 0,C 180,E1 10808.552,E2 10808.552} C_VEL
LIN {X 0,Y 218.81,Z 1174.328,A -85,B 0,C 180,E1 10802.881,E2 10802.881} C_VEL
LIN {X 0,Y 225.697,Z 1172.267,A -85,B 0,C 180,E1 10795.935,E2 10795.935} C_VEL
LIN {X 0,Y 236.699,Z 1168.344,A -85,B 0,C 180,E1 10788.548,E2 10788.548} C_VEL
LIN {X 0,Y 252.528,Z 1162.554,A -85,B 0,C 180,E1 10781.293,E2 10781.293} C_VEL
LIN {X 0,Y 275.165,Z 1154.062,A -85,B 0,C 180,E1 10774.147,E2 10774.147} C_VEL
LIN {X 0,Y 282.297,Z 1151.363,A -85,B 0,C 180,E1 10772.311,E2 10772.311} C_VEL
LIN {X 0,Y 254.932,Z 1174.711,A -85,B 0,C 180,E1 10764.666,E2 10764.666} C_VEL
LIN {X 0,Y 253.807,Z 1175.745,A -85,B 0,C 180,E1 10764.273,E2 10764.273} C_VEL
LIN {X 0,Y 249.357,Z 1179.291,A -85,B 0,C 180,E1 10763.059,E2 10763.059} C_VEL
LIN {X 0,Y 235.826,Z 1188.265,A -85,B 0,C 180,E1 10760.244,E2 10760.244} C_VEL
LIN {X 0,Y 231.749,Z 1191.497,A -85,B 0,C 180,E1 10758.846,E2 10758.846} C_VEL
LIN {X 0,Y 219.2,Z 1205.089,A -85,B 0,C 180,E1 10751.408,E2 10751.408} C_VEL
LIN {X 0,Y 210.069,Z 1216.983,A -85,B 0,C 180,E1 10743.099,E2 10743.099} C_VEL
LIN {X 0,Y 205.737,Z 1224.45,A -85,B 0,C 180,E1 10736.559,E2 10736.559} C_VEL
LIN {X 0,Y 203.496,Z 1230.127,A -85,B 0,C 180,E1 10730.417,E2 10730.417} C_VEL
LIN {X 0,Y 202.69,Z 1234.377,A -85,B 0,C 180,E1 10724.571,E2 10724.571} C_VEL
LIN {X 0,Y 202.818,Z 1237.335,A -85,B 0,C 180,E1 10719.077,E2 10719.077} C_VEL
LIN {X 0,Y 203.28,Z 1239.056,A -85,B 0,C 180,E1 10713.949,E2 10713.949} C_VEL
LIN {X 0,Y 203.385,Z 1239.62,A -85,B 0,C 180,E1 10709.437,E2 10709.437} C_VEL
LIN {X 0,Y 203.145,Z 1239.129,A -85,B 0,C 180,E1 10704.917,E2 10704.917} C_VEL
LIN {X 0,Y 202.661,Z 1237.235,A -85,B 0,C 180,E1 10699.062,E2 10699.062} C_VEL
LIN {X 0,Y 202.987,Z 1233.245,A -85,B 0,C 180,E1 10692.218,E2 10692.218} C_VEL
LIN {X 0,Y 204.698,Z 1228.045,A -85,B 0,C 180,E1 10685.986,E2 10685.986} C_VEL
LIN {X 0,Y 207.735,Z 1221.936,A -85,B 0,C 180,E1 10680.28,E2 10680.28} C_VEL
LIN {X 0,Y 212.142,Z 1214.814,A -85,B 0,C 180,E1 10674.899,E2 10674.899} C_VEL
LIN {X 0,Y 218.349,Z 1205.966,A -85,B 0,C 180,E1 10669.439,E2 10669.439} C_VEL
LIN {X 0,Y 228.384,Z 1192.777,A -85,B 0,C 180,E1 10663.019,E2 10663.019} C_VEL
LIN {X 0,Y 237.447,Z 1181.258,A -85,B 0,C 180,E1 10658.553,E2 10658.553} C_VEL
LIN {X 0,Y 247.476,Z 1168.582,A -85,B 0,C 180,E1 10654.49,E2 10654.49} C_VEL
LIN {X 0,Y 260.307,Z 1152.184,A -85,B 0,C 180,E1 10650.202,E2 10650.202} C_VEL
LIN {X 0,Y 273.366,Z 1134.64,A -85,B 0,C 180,E1 10646.567,E2 10646.567} C_VEL
LIN {X 0,Y 284.409,Z 1119.24,A -85,B 0,C 180,E1 10643.927,E2 10643.927} C_VEL
LIN {X 0,Y 297.178,Z 1100.537,A -85,B 0,C 180,E1 10641.253,E2 10641.253} C_VEL
LIN {X 0,Y 310.736,Z 1079.079,A -85,B 0,C 180,E1 10638.771,E2 10638.771} C_VEL
LIN {X 0,Y 321.947,Z 1059.96,A -85,B 0,C 180,E1 10636.95,E2 10636.95} C_VEL
LIN {X 0,Y 333.255,Z 1039.194,A -85,B 0,C 180,E1 10635.29,E2 10635.29} C_VEL
LIN {X 0,Y 346.169,Z 1013.113,A -85,B 0,C 180,E1 10633.604,E2 10633.604} C_VEL
LIN {X 0,Y 355.8,Z 991.5,A -85,B 0,C 180,E1 10632.47,E2 10632.47} C_VEL
LIN {X 0,Y 365.24,Z 968.141,A -85,B 0,C 180,E1 10631.463,E2 10631.463} C_VEL
LIN {X 0,Y 375.232,Z 939.789,A -85,B 0,C 180,E1 10630.496,E2 10630.496} C_VEL
LIN {X 0,Y 382.356,Z 916.27,A -85,B 0,C 180,E1 10629.865,E2 10629.865} C_VEL
LIN {X 0,Y 388.913,Z 890.182,A -85,B 0,C 180,E1 10629.248,E2 10629.248} C_VEL
LIN {X 0,Y 394.397,Z 861.215,A -85,B 0,C 180,E1 10628.663,E2 10628.663} C_VEL
LIN {X 0,Y 424.133,Z 651.687,A -85,B 0,C 180,E1 10625.214,E2 10625.214} C_VEL
LIN {X 0,Y 418.039,Z 640.844,A -85,B 0,C 180,E1 10621.988,E2 10621.988} C_VEL
LIN {X 0,Y 412.596,Z 631.533,A -85,B 0,C 180,E1 10618.75,E2 10618.75} C_VEL
LIN {X 0,Y 407.553,Z 623.266,A -85,B 0,C 180,E1 10615.356,E2 10615.356} C_VEL
LIN {X 0,Y 403.14,Z 616.212,A -85,B 0,C 180,E1 10611.944,E2 10611.944} C_VEL
LIN {X 0,Y 400.538,Z 612.159,A -85,B 0,C 180,E1 10609.645,E2 10609.645} C_VEL
LIN {X 0,Y 397.92,Z 607.862,A -85,B 0,C 180,E1 10607.003,E2 10607.003} C_VEL
LIN {X 0,Y 395.183,Z 603.359,A -85,B 0,C 180,E1 10603.84,E2 10603.84} C_VEL
LIN {X 0,Y 393.044,Z 600.169,A -85,B 0,C 180,E1 10600.996,E2 10600.996} C_VEL
LIN {X 0,Y 389.997,Z 597.091,A -85,B 0,C 180,E1 10596.103,E2 10596.103} C_VEL
LIN {X 0,Y 388.843,Z 594.55,A -85,B 0,C 180,E1 10592.925,E2 10592.925} C_VEL
LIN {X 0,Y 387.549,Z 593.929,A -85,B 0,C 180,E1 10588.589,E2 10588.589} C_VEL
LIN {X 0,Y 387.239,Z 593.617,A -85,B 0,C 180,E1 10583.669,E2 10583.669} C_VEL
LIN {X 0,Y 387.894,Z 593.998,A -85,B 0,C 180,E1 10579.049,E2 10579.049} C_VEL
LIN {X 0,Y 389.496,Z 594.95,A -85,B 0,C 180,E1 10574.78,E2 10574.78} C_VEL
LIN {X 0,Y 392.022,Z 598.99,A -85,B 0,C 180,E1 10569.849,E2 10569.849} C_VEL
LIN {X 0,Y 394.163,Z 600.803,A -85,B 0,C 180,E1 10567.138,E2 10567.138} C_VEL
LIN {X 0,Y 397.668,Z 605.398,A -85,B 0,C 180,E1 10563.239,E2 10563.239} C_VEL
LIN {X 0,Y 398.938,Z 607.038,A -85,B 0,C 180,E1 10562.012,E2 10562.012} C_VEL
LIN {X 0,Y 402.857,Z 612.086,A -85,B 0,C 180,E1 10558.702,E2 10558.702} C_VEL
LIN {X 0,Y 406.882,Z 617.369,A -85,B 0,C 180,E1 10555.783,E2 10555.783} C_VEL
LIN {X 0,Y 411.204,Z 623.31,A -85,B 0,C 180,E1 10553.005,E2 10553.005} C_VEL
LIN {X 0,Y 416.258,Z 630.379,A -85,B 0,C 180,E1 10550.123,E2 10550.123} C_VEL
LIN {X 0,Y 420.106,Z 636.296,A -85,B 0,C 180,E1 10548.115,E2 10548.115} C_VEL
LIN {X 0,Y 396.705,Z 801.63,A -85,B 0,C 180,E1 10545.43,E2 10545.43} C_VEL
LIN {X 0,Y 390.792,Z 832.744,A -85,B 0,C 180,E1 10544.733,E2 10544.733} C_VEL
LIN {X 0,Y 385.166,Z 856.346,A -85,B 0,C 180,E1 10544.057,E2 10544.057} C_VEL
LIN {X 0,Y 377.673,Z 883.015,A -85,B 0,C 180,E1 10543.128,E2 10543.128} C_VEL
LIN {X 0,Y 368.608,Z 909.823,A -85,B 0,C 180,E1 10541.971,E2 10541.971} C_VEL
LIN {X 0,Y 360.428,Z 931.191,A -85,B 0,C 180,E1 10540.869,E2 10540.869} C_VEL
LIN {X 0,Y 349.929,Z 955.772,A -85,B 0,C 180,E1 10539.374,E2 10539.374} C_VEL
LIN {X 0,Y 338.46,Z 979.256,A -85,B 0,C 180,E1 10537.639,E2 10537.639} C_VEL
LIN {X 0,Y 328.363,Z 998.174,A -85,B 0,C 180,E1 10535.996,E2 10535.996} C_VEL
LIN {X 0,Y 315.636,Z 1020.194,A -85,B 0,C 180,E1 10533.73,E2 10533.73} C_VEL
LIN {X 0,Y 303.042,Z 1039.82,A -85,B 0,C 180,E1 10531.259,E2 10531.259} C_VEL
LIN {X 0,Y 292.028,Z 1055.885,A -85,B 0,C 180,E1 10528.86,E2 10528.86} C_VEL
LIN {X 0,Y 281.14,Z 1070.879,A -85,B 0,C 180,E1 10526.218,E2 10526.218} C_VEL
LIN {X 0,Y 267.686,Z 1088.407,A -85,B 0,C 180,E1 10522.488,E2 10522.488} C_VEL
LIN {X 0,Y 255.947,Z 1102.762,A -85,B 0,C 180,E1 10518.687,E2 10518.687} C_VEL
LIN {X 0,Y 245.995,Z 1114.559,A -85,B 0,C 180,E1 10514.922,E2 10514.922} C_VEL
LIN {X 0,Y 236.042,Z 1126.158,A -85,B 0,C 180,E1 10510.449,E2 10510.449} C_VEL
LIN {X 0,Y 225.554,Z 1138.318,A -85,B 0,C 180,E1 10504.533,E2 10504.533} C_VEL
LIN {X 0,Y 218.465,Z 1146.766,A -85,B 0,C 180,E1 10499.368,E2 10499.368} C_VEL
LIN {X 0,Y 212.88,Z 1153.89,A -85,B 0,C 180,E1 10494.048,E2 10494.048} C_VEL
LIN {X 0,Y 208.145,Z 1160.75,A -85,B 0,C 180,E1 10487.714,E2 10487.714} C_VEL
LIN {X 0,Y 204.9,Z 1166.692,A -85,B 0,C 180,E1 10480.426,E2 10480.426} C_VEL
LIN {X 0,Y 203.7,Z 1170.121,A -85,B 0,C 180,E1 10474.942,E2 10474.942} C_VEL
LIN {X 0,Y 203.317,Z 1172.762,A -85,B 0,C 180,E1 10469.458,E2 10469.458} C_VEL
LIN {X 0,Y 203.425,Z 1174.699,A -85,B 0,C 180,E1 10464.077,E2 10464.077} C_VEL
LIN {X 0,Y 204.032,Z 1175.981,A -85,B 0,C 180,E1 10458.871,E2 10458.871} C_VEL
LIN {X 0,Y 205.475,Z 1176.725,A -85,B 0,C 180,E1 10452.935,E2 10452.935} C_VEL
LIN {X 0,Y 208.35,Z 1176.702,A -85,B 0,C 180,E1 10446.59,E2 10446.59} C_VEL
LIN {X 0,Y 213.584,Z 1175.719,A -85,B 0,C 180,E1 10439.732,E2 10439.732} C_VEL
LIN {X 0,Y 222.832,Z 1173.089,A -85,B 0,C 180,E1 10432.004,E2 10432.004} C_VEL
LIN {X 0,Y 235.782,Z 1169.044,A -85,B 0,C 180,E1 10424.756,E2 10424.756} C_VEL
LIN {X 0,Y 255.431,Z 1162.438,A -85,B 0,C 180,E1 10417.199,E2 10417.199} C_VEL
LIN {X 0,Y 272.444,Z 1156.834,A -85,B 0,C 180,E1 10412.456,E2 10412.456} C_VEL
LIN {X 0,Y 244.751,Z 1179.209,A -85,B 0,C 180,E1 10404.387,E2 10404.387} C_VEL
LIN {X 0,Y 231.749,Z 1191.497,A -85,B 0,C 180,E1 10398.846,E2 10398.846} C_VEL
LIN {X 0,Y 227.784,Z 1194.79,A -85,B 0,C 180,E1 10397.388,E2 10397.388} C_VEL
LIN {X 0,Y 214.667,Z 1202.974,A -85,B 0,C 180,E1 10393.622,E2 10393.622} C_VEL
LIN {X 0,Y 211.712,Z 1205.367,A -85,B 0,C 180,E1 10392.153,E2 10392.153} C_VEL
LIN {X 0,Y 203.052,Z 1215.715,A -85,B 0,C 180,E1 10384.492,E2 10384.492} C_VEL
LIN {X 0,Y 198.4,Z 1222.891,A -85,B 0,C 180,E1 10377.949,E2 10377.949} C_VEL
LIN {X 0,Y 195.824,Z 1228.489,A -85,B 0,C 180,E1 10371.672,E2 10371.672} C_VEL
LIN {X 0,Y 194.817,Z 1232.845,A -85,B 0,C 180,E1 10365.479,E2 10365.479} C_VEL
LIN {X 0,Y 194.869,Z 1235.821,A -85,B 0,C 180,E1 10359.748,E2 10359.748} C_VEL
LIN {X 0,Y 195.354,Z 1237.605,A -85,B 0,C 180,E1 10354.403,E2 10354.403} C_VEL
LIN {X 0,Y 195.531,Z 1238.196,A -85,B 0,C 180,E1 10350,E2 10350} C_VEL
LIN {X 0,Y 195.302,Z 1237.777,A -85,B 0,C 180,E1 10345.301,E2 10345.301} C_VEL
LIN {X 0,Y 194.8,Z 1236.112,A -85,B 0,C 180,E1 10339.651,E2 10339.651} C_VEL
LIN {X 0,Y 194.993,Z 1232.498,A -85,B 0,C 180,E1 10332.698,E2 10332.698} C_VEL
LIN {X 0,Y 196.825,Z 1226.977,A -85,B 0,C 180,E1 10325.702,E2 10325.702} C_VEL
LIN {X 0,Y 199.876,Z 1221.091,A -85,B 0,C 180,E1 10319.934,E2 10319.934} C_VEL
LIN {X 0,Y 204.386,Z 1214.091,A -85,B 0,C 180,E1 10314.397,E2 10314.397} C_VEL
LIN {X 0,Y 210.348,Z 1205.895,A -85,B 0,C 180,E1 10309.096,E2 10309.096} C_VEL
LIN {X 0,Y 218.909,Z 1195.125,A -85,B 0,C 180,E1 10303.428,E2 10303.428} C_VEL
LIN {X 0,Y 230.134,Z 1181.311,A -85,B 0,C 180,E1 10297.745,E2 10297.745} C_VEL
LIN {X 0,Y 240.479,Z 1168.693,A -85,B 0,C 180,E1 10293.573,E2 10293.573} C_VEL
LIN {X 0,Y 252.065,Z 1154.371,A -85,B 0,C 180,E1 10289.69,E2 10289.69} C_VEL
LIN {X 0,Y 266.753,Z 1135.409,A -85,B 0,C 180,E1 10285.601,E2 10285.601} C_VEL
LIN {X 0,Y 278.714,Z 1119.156,A -85,B 0,C 180,E1 10282.783,E2 10282.783} C_VEL
LIN {X 0,Y 290.55,Z 1102.229,A -85,B 0,C 180,E1 10280.339,E2 10280.339} C_VEL
LIN {X 0,Y 305.369,Z 1079.518,A -85,B 0,C 180,E1 10277.669,E2 10277.669} C_VEL
LIN {X 0,Y 317.315,Z 1059.593,A -85,B 0,C 180,E1 10275.776,E2 10275.776} C_VEL
LIN {X 0,Y 328.469,Z 1039.533,A -85,B 0,C 180,E1 10274.181,E2 10274.181} C_VEL
LIN {X 0,Y 341.623,Z 1013.631,A -85,B 0,C 180,E1 10272.509,E2 10272.509} C_VEL
LIN {X 0,Y 351.828,Z 991.153,A -85,B 0,C 180,E1 10271.342,E2 10271.342} C_VEL
LIN {X 0,Y 361.317,Z 968.084,A -85,B 0,C 180,E1 10270.363,E2 10270.363} C_VEL
LIN {X 0,Y 371.688,Z 939.186,A -85,B 0,C 180,E1 10269.393,E2 10269.393} C_VEL
LIN {X 0,Y 378.89,Z 915.766,A -85,B 0,C 180,E1 10268.777,E2 10268.777} C_VEL
LIN {X 0,Y 385.316,Z 890.671,A -85,B 0,C 180,E1 10268.192,E2 10268.192} C_VEL
LIN {X 0,Y 391.103,Z 861.061,A -85,B 0,C 180,E1 10267.597,E2 10267.597} C_VEL
LIN {X 0,Y 414.576,Z 698.739,A -85,B 0,C 180,E1 10264.93,E2 10264.93} C_VEL
LIN {X 0,Y 420.711,Z 656.755,A -85,B 0,C 180,E1 10264.259,E2 10264.259} C_VEL
LIN {X 0,Y 414.702,Z 646.122,A -85,B 0,C 180,E1 10260.967,E2 10260.967} C_VEL
LIN {X 0,Y 409.917,Z 637.991,A -85,B 0,C 180,E1 10258.043,E2 10258.043} C_VEL
LIN {X 0,Y 405.095,Z 629.882,A -85,B 0,C 180,E1 10254.689,E2 10254.689} C_VEL
LIN {X 0,Y 399.997,Z 621.481,A -85,B 0,C 180,E1 10250.504,E2 10250.504} C_VEL
LIN {X 0,Y 396.071,Z 615.425,A -85,B 0,C 180,E1 10246.719,E2 10246.719} C_VEL
LIN {X 0,Y 393.583,Z 611.202,A -85,B 0,C 180,E1 10243.772,E2 10243.772} C_VEL
LIN {X 0,Y 391.437,Z 607.988,A -85,B 0,C 180,E1 10240.915,E2 10240.915} C_VEL
LIN {X 0,Y 388.375,Z 604.891,A -85,B 0,C 180,E1 10235.997,E2 10235.997} C_VEL
LIN {X 0,Y 387.227,Z 602.361,A -85,B 0,C 180,E1 10232.803,E2 10232.803} C_VEL
LIN {X 0,Y 385.963,Z 601.761,A -85,B 0,C 180,E1 10228.445,E2 10228.445} C_VEL
LIN {X 0,Y 385.675,Z 601.487,A -85,B 0,C 180,E1 10223.395,E2 10223.395} C_VEL
LIN {X 0,Y 386.402,Z 601.872,A -85,B 0,C 180,E1 10218.852,E2 10218.852} C_VEL
LIN {X 0,Y 387.88,Z 602.714,A -85,B 0,C 180,E1 10214.936,E2 10214.936} C_VEL
LIN {X 0,Y 390.264,Z 606.623,A -85,B 0,C 180,E1 10210.213,E2 10210.213} C_VEL
LIN {X 0,Y 392.574,Z 608.682,A -85,B 0,C 180,E1 10207.213,E2 10207.213} C_VEL
LIN {X 0,Y 396.199,Z 613.327,A -85,B 0,C 180,E1 10203.205,E2 10203.205} C_VEL
LIN {X 0,Y 401.074,Z 619.732,A -85,B 0,C 180,E1 10198.923,E2 10198.923} C_VEL
LIN {X 0,Y 405.217,Z 625.234,A -85,B 0,C 180,E1 10195.897,E2 10195.897} C_VEL
LIN {X 0,Y 409.544,Z 631.223,A -85,B 0,C 180,E1 10193.096,E2 10193.096} C_VEL
LIN {X 0,Y 414.871,Z 638.845,A -85,B 0,C 180,E1 10190.05,E2 10190.05} C_VEL
LIN {X 0,Y 416.71,Z 641.732,A -85,B 0,C 180,E1 10189.069,E2 10189.069} C_VEL
LIN {X 0,Y 393.36,Z 803.239,A -85,B 0,C 180,E1 10186.473,E2 10186.473} C_VEL
LIN {X 0,Y 387.357,Z 834.074,A -85,B 0,C 180,E1 10185.786,E2 10185.786} C_VEL
LIN {X 0,Y 381.358,Z 858.699,A -85,B 0,C 180,E1 10185.083,E2 10185.083} C_VEL
LIN {X 0,Y 373.21,Z 886.731,A -85,B 0,C 180,E1 10184.102,E2 10184.102} C_VEL
LIN {X 0,Y 364.704,Z 911.315,A -85,B 0,C 180,E1 10183.044,E2 10183.044} C_VEL
LIN {X 0,Y 355.916,Z 933.85,A -85,B 0,C 180,E1 10181.89,E2 10181.89} C_VEL
LIN {X 0,Y 344.206,Z 960.333,A -85,B 0,C 180,E1 10180.261,E2 10180.261} C_VEL
LIN {X 0,Y 333.822,Z 981.189,A -85,B 0,C 180,E1 10178.717,E2 10178.717} C_VEL
LIN {X 0,Y 323.42,Z 1000.318,A -85,B 0,C 180,E1 10177.061,E2 10177.061} C_VEL
LIN {X 0,Y 310.021,Z 1022.865,A -85,B 0,C 180,E1 10174.725,E2 10174.725} C_VEL
LIN {X 0,Y 297.496,Z 1041.937,A -85,B 0,C 180,E1 10172.312,E2 10172.312} C_VEL
LIN {X 0,Y 286.315,Z 1057.852,A -85,B 0,C 180,E1 10169.922,E2 10169.922} C_VEL
LIN {X 0,Y 272.762,Z 1076.059,A -85,B 0,C 180,E1 10166.638,E2 10166.638} C_VEL
LIN {X 0,Y 259.415,Z 1092.556,A -85,B 0,C 180,E1 10162.915,E2 10162.915} C_VEL
LIN {X 0,Y 249.093,Z 1104.827,A -85,B 0,C 180,E1 10159.567,E2 10159.567} C_VEL
LIN {X 0,Y 239.217,Z 1116.187,A -85,B 0,C 180,E1 10155.867,E2 10155.867} C_VEL
LIN {X 0,Y 227.961,Z 1128.974,A -85,B 0,C 180,E1 10150.794,E2 10150.794} C_VEL
LIN {X 0,Y 217.808,Z 1140.255,A -85,B 0,C 180,E1 10145.018,E2 10145.018} C_VEL
LIN {X 0,Y 211.065,Z 1148.045,A -85,B 0,C 180,E1 10140.105,E2 10140.105} C_VEL
LIN {X 0,Y 205.466,Z 1154.916,A -85,B 0,C 180,E1 10134.842,E2 10134.842} C_VEL
LIN {X 0,Y 200.996,Z 1161.02,A -85,B 0,C 180,E1 10129.126,E2 10129.126} C_VEL
LIN {X 0,Y 197.458,Z 1167.141,A -85,B 0,C 180,E1 10121.895,E2 10121.895} C_VEL
LIN {X 0,Y 195.83,Z 1171.281,A -85,B 0,C 180,E1 10115.222,E2 10115.222} C_VEL
LIN {X 0,Y 195.418,Z 1174.065,A -85,B 0,C 180,E1 10109.42,E2 10109.42} C_VEL
LIN {X 0,Y 195.554,Z 1176.086,A -85,B 0,C 180,E1 10103.762,E2 10103.762} C_VEL
LIN {X 0,Y 196.273,Z 1177.484,A -85,B 0,C 180,E1 10098.105,E2 10098.105} C_VEL
LIN {X 0,Y 197.925,Z 1178.305,A -85,B 0,C 180,E1 10091.954,E2 10091.954} C_VEL
LIN {X 0,Y 201.155,Z 1178.379,A -85,B 0,C 180,E1 10085.419,E2 10085.419} C_VEL
LIN {X 0,Y 207.236,Z 1177.468,A -85,B 0,C 180,E1 10078.065,E2 10078.065} C_VEL
LIN {X 0,Y 217.743,Z 1174.878,A -85,B 0,C 180,E1 10069.951,E2 10069.951} C_VEL
LIN {X 0,Y 232.863,Z 1170.769,A -85,B 0,C 180,E1 10062.25,E2 10062.25} C_VEL
LIN {X 0,Y 258.048,Z 1163.269,A -85,B 0,C 180,E1 10053.786,E2 10053.786} C_VEL
LIN {X 0,Y 262.442,Z 1161.885,A -85,B 0,C 180,E1 10052.586,E2 10052.586} C_VEL
LIN {X 0,Y 233.458,Z 1184.491,A -85,B 0,C 180,E1 10043.628,E2 10043.628} C_VEL
LIN {X 0,Y 218.259,Z 1198.475,A -85,B 0,C 180,E1 10036.37,E2 10036.37} C_VEL
LIN {X 0,Y 211.712,Z 1205.367,A -85,B 0,C 180,E1 10032.153,E2 10032.153} C_VEL
LIN {X 0,Y 208.292,Z 1208.106,A -85,B 0,C 180,E1 10030.392,E2 10030.392} C_VEL
LIN {X 0,Y 196.666,Z 1214.779,A -85,B 0,C 180,E1 10025.72,E2 10025.72} C_VEL
LIN {X 0,Y 194.374,Z 1216.778,A -85,B 0,C 180,E1 10023.988,E2 10023.988} C_VEL
LIN {X 0,Y 188.967,Z 1225.328,A -85,B 0,C 180,E1 10015.043,E2 10015.043} C_VEL
LIN {X 0,Y 187.01,Z 1230.944,A -85,B 0,C 180,E1 10007.101,E2 10007.101} C_VEL
LIN {X 0,Y 186.892,Z 1234.2,A -85,B 0,C 180,E1 10000.792,E2 10000.792} C_VEL
LIN {X 0,Y 187.422,Z 1236.129,A -85,B 0,C 180,E1 9994.896,E2 9994.896} C_VEL
LIN {X 0,Y 187.641,Z 1236.79,A -85,B 0,C 180,E1 9990.305,E2 9990.305} C_VEL
LIN {X 0,Y 187.461,Z 1236.433,A -85,B 0,C 180,E1 9985.717,E2 9985.717} C_VEL
LIN {X 0,Y 186.941,Z 1234.933,A -85,B 0,C 180,E1 9980.145,E2 9980.145} C_VEL
LIN {X 0,Y 186.968,Z 1231.974,A -85,B 0,C 180,E1 9973.854,E2 9973.854} C_VEL
LIN {X 0,Y 188.619,Z 1226.637,A -85,B 0,C 180,E1 9966.242,E2 9966.242} C_VEL
LIN {X 0,Y 191.965,Z 1220.327,A -85,B 0,C 180,E1 9959.653,E2 9959.653} C_VEL
LIN {X 0,Y 196.943,Z 1212.961,A -85,B 0,C 180,E1 9953.558,E2 9953.558} C_VEL
LIN {X 0,Y 203.284,Z 1204.671,A -85,B 0,C 180,E1 9948.015,E2 9948.015} C_VEL
LIN {X 0,Y 212.587,Z 1193.497,A -85,B 0,C 180,E1 9942.001,E2 9942.001} C_VEL
LIN {X 0,Y 223.886,Z 1180.115,A -85,B 0,C 180,E1 9936.441,E2 9936.441} C_VEL
LIN {X 0,Y 234.3,Z 1167.837,A -85,B 0,C 180,E1 9932.332,E2 9932.332} C_VEL
LIN {X 0,Y 245.167,Z 1154.794,A -85,B 0,C 180,E1 9928.736,E2 9928.736} C_VEL
LIN {X 0,Y 259.05,Z 1137.616,A -85,B 0,C 180,E1 9924.88,E2 9924.88} C_VEL
LIN {X 0,Y 273.133,Z 1118.993,A -85,B 0,C 180,E1 9921.591,E2 9921.591} C_VEL
LIN {X 0,Y 284.846,Z 1102.684,A -85,B 0,C 180,E1 9919.221,E2 9919.221} C_VEL
LIN {X 0,Y 298.981,Z 1081.776,A -85,B 0,C 180,E1 9916.715,E2 9916.715} C_VEL
LIN {X 0,Y 312.519,Z 1059.741,A -85,B 0,C 180,E1 9914.611,E2 9914.611} C_VEL
LIN {X 0,Y 323.944,Z 1039.632,A -85,B 0,C 180,E1 9913.022,E2 9913.022} C_VEL
LIN {X 0,Y 336.657,Z 1015.309,A -85,B 0,C 180,E1 9911.448,E2 9911.448} C_VEL
LIN {X 0,Y 347.951,Z 990.921,A -85,B 0,C 180,E1 9910.195,E2 9910.195} C_VEL
LIN {X 0,Y 357.127,Z 969.027,A -85,B 0,C 180,E1 9909.277,E2 9909.277} C_VEL
LIN {X 0,Y 367.208,Z 941.887,A -85,B 0,C 180,E1 9908.361,E2 9908.361} C_VEL
LIN {X 0,Y 375.329,Z 916.096,A -85,B 0,C 180,E1 9907.69,E2 9907.69} C_VEL
LIN {X 0,Y 381.748,Z 891.589,A -85,B 0,C 180,E1 9907.126,E2 9907.126} C_VEL
LIN {X 0,Y 388.03,Z 860.468,A -85,B 0,C 180,E1 9906.505,E2 9906.505} C_VEL
LIN {X 0,Y 417.395,Z 661.928,A -85,B 0,C 180,E1 9903.305,E2 9903.305} C_VEL
LIN {X 0,Y 411.681,Z 651.855,A -85,B 0,C 180,E1 9900.07,E2 9900.07} C_VEL
LIN {X 0,Y 407.207,Z 644.246,A -85,B 0,C 180,E1 9897.255,E2 9897.255} C_VEL
LIN {X 0,Y 402.761,Z 636.758,A -85,B 0,C 180,E1 9894.086,E2 9894.086} C_VEL
LIN {X 0,Y 398.161,Z 629.066,A -85,B 0,C 180,E1 9890.241,E2 9890.241} C_VEL
LIN {X 0,Y 394.282,Z 623.088,A -85,B 0,C 180,E1 9886.508,E2 9886.508} C_VEL
LIN {X 0,Y 391.82,Z 618.87,A -85,B 0,C 180,E1 9883.545,E2 9883.545} C_VEL
LIN {X 0,Y 389.722,Z 615.726,A -85,B 0,C 180,E1 9880.672,E2 9880.672} C_VEL
LIN {X 0,Y 386.678,Z 612.567,A -85,B 0,C 180,E1 9875.723,E2 9875.723} C_VEL
LIN {X 0,Y 385.653,Z 610.205,A -85,B 0,C 180,E1 9872.784,E2 9872.784} C_VEL
LIN {X 0,Y 384.377,Z 609.589,A -85,B 0,C 180,E1 9868.279,E2 9868.279} C_VEL
LIN {X 0,Y 384.117,Z 609.355,A -85,B 0,C 180,E1 9863.222,E2 9863.222} C_VEL
LIN {X 0,Y 384.915,Z 609.745,A -85,B 0,C 180,E1 9858.653,E2 9858.653} C_VEL
LIN {X 0,Y 386.316,Z 610.623,A -85,B 0,C 180,E1 9854.958,E2 9854.958} C_VEL
LIN {X 0,Y 388.887,Z 614.654,A -85,B 0,C 180,E1 9849.985,E2 9849.985} C_VEL
LIN {X 0,Y 390.974,Z 616.531,A -85,B 0,C 180,E1 9847.308,E2 9847.308} C_VEL
LIN {X 0,Y 394.626,Z 621.169,A -85,B 0,C 180,E1 9843.264,E2 9843.264} C_VEL
LIN {X 0,Y 399.357,Z 627.472,A -85,B 0,C 180,E1 9839.095,E2 9839.095} C_VEL
LIN {X 0,Y 403.384,Z 632.883,A -85,B 0,C 180,E1 9836.11,E2 9836.11} C_VEL
LIN {X 0,Y 408.136,Z 639.459,A -85,B 0,C 180,E1 9833.036,E2 9833.036} C_VEL
LIN {X 0,Y 413.377,Z 647.116,A -85,B 0,C 180,E1 9830.038,E2 9830.038} C_VEL
LIN {X 0,Y 390.303,Z 803.822,A -85,B 0,C 180,E1 9827.55,E2 9827.55} C_VEL
LIN {X 0,Y 384.184,Z 834.83,A -85,B 0,C 180,E1 9826.872,E2 9826.872} C_VEL
LIN {X 0,Y 378.172,Z 859.135,A -85,B 0,C 180,E1 9826.189,E2 9826.189} C_VEL
LIN {X 0,Y 370.218,Z 886.339,A -85,B 0,C 180,E1 9825.26,E2 9825.26} C_VEL
LIN {X 0,Y 360.892,Z 912.862,A -85,B 0,C 180,E1 9824.136,E2 9824.136} C_VEL
LIN {X 0,Y 351.801,Z 935.733,A -85,B 0,C 180,E1 9822.975,E2 9822.975} C_VEL
LIN {X 0,Y 339.571,Z 962.719,A -85,B 0,C 180,E1 9821.32,E2 9821.32} C_VEL
LIN {X 0,Y 329.085,Z 983.338,A -85,B 0,C 180,E1 9819.796,E2 9819.796} C_VEL
LIN {X 0,Y 317.401,Z 1004.344,A -85,B 0,C 180,E1 9817.967,E2 9817.967} C_VEL
LIN {X 0,Y 303.957,Z 1026.177,A -85,B 0,C 180,E1 9815.664,E2 9815.664} C_VEL
LIN {X 0,Y 292.179,Z 1043.741,A -85,B 0,C 180,E1 9813.434,E2 9813.434} C_VEL
LIN {X 0,Y 280.666,Z 1059.783,A -85,B 0,C 180,E1 9811.021,E2 9811.021} C_VEL
LIN {X 0,Y 266.46,Z 1078.341,A -85,B 0,C 180,E1 9807.634,E2 9807.634} C_VEL
LIN {X 0,Y 253.347,Z 1094.171,A -85,B 0,C 180,E1 9804.032,E2 9804.032} C_VEL
LIN {X 0,Y 242.301,Z 1106.927,A -85,B 0,C 180,E1 9800.496,E2 9800.496} C_VEL
LIN {X 0,Y 229.977,Z 1120.716,A -85,B 0,C 180,E1 9795.827,E2 9795.827} C_VEL
LIN {X 0,Y 218.243,Z 1133.354,A -85,B 0,C 180,E1 9790.317,E2 9790.317} C_VEL
LIN {X 0,Y 209.953,Z 1142.351,A -85,B 0,C 180,E1 9785.455,E2 9785.455} C_VEL
LIN {X 0,Y 202.776,Z 1150.406,A -85,B 0,C 180,E1 9780.131,E2 9780.131} C_VEL
LIN {X 0,Y 195.948,Z 1158.791,A -85,B 0,C 180,E1 9773.24,E2 9773.24} C_VEL
LIN {X 0,Y 191.22,Z 1165.461,A -85,B 0,C 180,E1 9765.937,E2 9765.937} C_VEL
LIN {X 0,Y 188.866,Z 1169.867,A -85,B 0,C 180,E1 9759.837,E2 9759.837} C_VEL
LIN {X 0,Y 187.82,Z 1173.021,A -85,B 0,C 180,E1 9754.355,E2 9754.355} C_VEL
LIN {X 0,Y 187.503,Z 1175.477,A -85,B 0,C 180,E1 9749.009,E2 9749.009} C_VEL
LIN {X 0,Y 187.687,Z 1177.53,A -85,B 0,C 180,E1 9743.218,E2 9743.218} C_VEL
LIN {X 0,Y 188.537,Z 1179.006,A -85,B 0,C 180,E1 9737.277,E2 9737.277} C_VEL
LIN {X 0,Y 190.423,Z 1179.91,A -85,B 0,C 180,E1 9730.896,E2 9730.896} C_VEL
LIN {X 0,Y 194.068,Z 1180.077,A -85,B 0,C 180,E1 9724.137,E2 9724.137} C_VEL
LIN {X 0,Y 201.68,Z 1179.2,A -85,B 0,C 180,E1 9715.735,E2 9715.735} C_VEL
LIN {X 0,Y 213.855,Z 1176.543,A -85,B 0,C 180,E1 9707.306,E2 9707.306} C_VEL
LIN {X 0,Y 231.011,Z 1172.361,A -85,B 0,C 180,E1 9699.476,E2 9699.476} C_VEL
LIN {X 0,Y 252.432,Z 1166.746,A -85,B 0,C 180,E1 9692.708,E2 9692.708} C_VEL
LIN {X 0,Y 226.14,Z 1186.051,A -85,B 0,C 180,E1 9684.444,E2 9684.444} C_VEL
LIN {X 0,Y 208.301,Z 1201.681,A -85,B 0,C 180,E1 9675.661,E2 9675.661} C_VEL
LIN {X 0,Y 197.249,Z 1213.198,A -85,B 0,C 180,E1 9667.101,E2 9667.101} C_VEL
LIN {X 0,Y 194.374,Z 1216.778,A -85,B 0,C 180,E1 9663.988,E2 9663.988} C_VEL
LIN {X 0,Y 191.771,Z 1219.016,A -85,B 0,C 180,E1 9661.922,E2 9661.922} C_VEL
LIN {X 0,Y 182.043,Z 1224.1,A -85,B 0,C 180,E1 9656.126,E2 9656.126} C_VEL
LIN {X 0,Y 180.659,Z 1225.389,A -85,B 0,C 180,E1 9654.288,E2 9654.288} C_VEL
LIN {X 0,Y 179.142,Z 1229.573,A -85,B 0,C 180,E1 9647.877,E2 9647.877} C_VEL
LIN {X 0,Y 178.932,Z 1232.672,A -85,B 0,C 180,E1 9641.605,E2 9641.605} C_VEL
LIN {X 0,Y 179.466,Z 1234.659,A -85,B 0,C 180,E1 9635.435,E2 9635.435} C_VEL
LIN {X 0,Y 179.762,Z 1235.364,A -85,B 0,C 180,E1 9630.637,E2 9630.637} C_VEL
LIN {X 0,Y 179.597,Z 1235.02,A -85,B 0,C 180,E1 9625.849,E2 9625.849} C_VEL
LIN {X 0,Y 179.047,Z 1233.516,A -85,B 0,C 180,E1 9620.031,E2 9620.031} C_VEL
LIN {X 0,Y 179.122,Z 1230.381,A -85,B 0,C 180,E1 9613.126,E2 9613.126} C_VEL
LIN {X 0,Y 181.053,Z 1224.872,A -85,B 0,C 180,E1 9605.183,E2 9605.183} C_VEL
LIN {X 0,Y 184.528,Z 1218.804,A -85,B 0,C 180,E1 9598.656,E2 9598.656} C_VEL
LIN {X 0,Y 189.544,Z 1211.785,A -85,B 0,C 180,E1 9592.653,E2 9592.653} C_VEL
LIN {X 0,Y 195.807,Z 1203.956,A -85,B 0,C 180,E1 9587.222,E2 9587.222} C_VEL
LIN {X 0,Y 204.153,Z 1194.27,A -85,B 0,C 180,E1 9581.766,E2 9581.766} C_VEL
LIN {X 0,Y 216.564,Z 1180.22,A -85,B 0,C 180,E1 9575.574,E2 9575.574} C_VEL
LIN {X 0,Y 227.849,Z 1167.379,A -85,B 0,C 180,E1 9571.16,E2 9571.16} C_VEL
LIN {X 0,Y 239.024,Z 1154.409,A -85,B 0,C 180,E1 9567.522,E2 9567.522} C_VEL
LIN {X 0,Y 253.238,Z 1137.372,A -85,B 0,C 180,E1 9563.649,E2 9563.649} C_VEL
LIN {X 0,Y 267.843,Z 1118.612,A -85,B 0,C 180,E1 9560.315,E2 9560.315} C_VEL
LIN {X 0,Y 279.635,Z 1102.586,A -85,B 0,C 180,E1 9557.988,E2 9557.988} C_VEL
LIN {X 0,Y 292.873,Z 1083.429,A -85,B 0,C 180,E1 9555.687,E2 9555.687} C_VEL
LIN {X 0,Y 307.856,Z 1059.751,A -85,B 0,C 180,E1 9553.41,E2 9553.41} C_VEL
LIN {X 0,Y 319.282,Z 1040.025,A -85,B 0,C 180,E1 9551.865,E2 9551.865} C_VEL
LIN {X 0,Y 331.405,Z 1017.338,A -85,B 0,C 180,E1 9550.401,E2 9550.401} C_VEL
LIN {X 0,Y 343.536,Z 991.884,A -85,B 0,C 180,E1 9549.089,E2 9549.089} C_VEL
LIN {X 0,Y 353.141,Z 969.401,A -85,B 0,C 180,E1 9548.158,E2 9548.158} C_VEL
LIN {X 0,Y 363.178,Z 943.074,A -85,B 0,C 180,E1 9547.276,E2 9547.276} C_VEL
LIN {X 0,Y 371.904,Z 915.883,A -85,B 0,C 180,E1 9546.58,E2 9546.58} C_VEL
LIN {X 0,Y 378.154,Z 892.52,A -85,B 0,C 180,E1 9546.052,E2 9546.052} C_VEL
LIN {X 0,Y 384.327,Z 863.528,A -85,B 0,C 180,E1 9545.469,E2 9545.469} C_VEL
LIN {X 0,Y 393.229,Z 805.385,A -85,B 0,C 180,E1 9544.506,E2 9544.506} C_VEL
LIN {X 0,Y 413.888,Z 667.063,A -85,B 0,C 180,E1 9542.319,E2 9542.319} C_VEL
LIN {X 0,Y 408.97,Z 658.253,A -85,B 0,C 180,E1 9539.425,E2 9539.425} C_VEL
LIN {X 0,Y 404.56,Z 650.612,A -85,B 0,C 180,E1 9536.528,E2 9536.528} C_VEL
LIN {X 0,Y 400.113,Z 643.135,A -85,B 0,C 180,E1 9533.255,E2 9533.255} C_VEL
LIN {X 0,Y 396.068,Z 636.399,A -85,B 0,C 180,E1 9529.821,E2 9529.821} C_VEL
LIN {X 0,Y 392.661,Z 630.966,A -85,B 0,C 180,E1 9526.451,E2 9526.451} C_VEL
LIN {X 0,Y 390.043,Z 626.532,A -85,B 0,C 180,E1 9523.314,E2 9523.314} C_VEL
LIN {X 0,Y 388.093,Z 623.527,A -85,B 0,C 180,E1 9520.554,E2 9520.554} C_VEL
LIN {X 0,Y 385.061,Z 620.368,A -85,B 0,C 180,E1 9515.614,E2 9515.614} C_VEL
LIN {X 0,Y 384.015,Z 618.021,A -85,B 0,C 180,E1 9512.607,E2 9512.607} C_VEL
LIN {X 0,Y 382.783,Z 617.398,A -85,B 0,C 180,E1 9507.976,E2 9507.976} C_VEL
LIN {X 0,Y 382.563,Z 617.221,A -85,B 0,C 180,E1 9503.048,E2 9503.048} C_VEL
LIN {X 0,Y 383.432,Z 617.619,A -85,B 0,C 180,E1 9498.453,E2 9498.453} C_VEL
LIN {X 0,Y 384.674,Z 618.295,A -85,B 0,C 180,E1 9495.203,E2 9495.203} C_VEL
LIN {X 0,Y 387.076,Z 622.24,A -85,B 0,C 180,E1 9490.419,E2 9490.419} C_VEL
LIN {X 0,Y 389.327,Z 624.278,A -85,B 0,C 180,E1 9487.477,E2 9487.477} C_VEL
LIN {X 0,Y 392.948,Z 628.921,A -85,B 0,C 180,E1 9483.423,E2 9483.423} C_VEL
LIN {X 0,Y 397.593,Z 635.176,A -85,B 0,C 180,E1 9479.284,E2 9479.284} C_VEL
LIN {X 0,Y 401.47,Z 640.403,A -85,B 0,C 180,E1 9476.387,E2 9476.387} C_VEL
LIN {X 0,Y 406.153,Z 646.936,A -85,B 0,C 180,E1 9473.324,E2 9473.324} C_VEL
LIN {X 0,Y 410.121,Z 652.682,A -85,B 0,C 180,E1 9471.015,E2 9471.015} C_VEL
LIN {X 0,Y 387.353,Z 804.406,A -85,B 0,C 180,E1 9468.643,E2 9468.643} C_VEL
LIN {X 0,Y 381.122,Z 835.535,A -85,B 0,C 180,E1 9467.974,E2 9467.974} C_VEL
LIN {X 0,Y 375.185,Z 859.269,A -85,B 0,C 180,E1 9467.321,E2 9467.321} C_VEL
LIN {X 0,Y 367.409,Z 885.684,A -85,B 0,C 180,E1 9466.441,E2 9466.441} C_VEL
LIN {X 0,Y 357.953,Z 912.477,A -85,B 0,C 180,E1 9465.338,E2 9465.338} C_VEL
LIN {X 0,Y 349.179,Z 934.374,A -85,B 0,C 180,E1 9464.256,E2 9464.256} C_VEL
LIN {X 0,Y 337.927,Z 959.423,A -85,B 0,C 180,E1 9462.787,E2 9462.787} C_VEL
LIN {X 0,Y 326.063,Z 982.547,A -85,B 0,C 180,E1 9461.139,E2 9461.139} C_VEL
LIN {X 0,Y 315.111,Z 1002.033,A -85,B 0,C 180,E1 9459.497,E2 9459.497} C_VEL
LIN {X 0,Y 301.369,Z 1024.41,A -85,B 0,C 180,E1 9457.236,E2 9457.236} C_VEL
LIN {X 0,Y 288.567,Z 1043.23,A -85,B 0,C 180,E1 9454.909,E2 9454.909} C_VEL
LIN {X 0,Y 277.264,Z 1058.747,A -85,B 0,C 180,E1 9452.632,E2 9452.632} C_VEL
LIN {X 0,Y 265.561,Z 1073.857,A -85,B 0,C 180,E1 9450,E2 9450} C_VEL
LIN {X 0,Y 251.029,Z 1091.492,A -85,B 0,C 180,E1 9446.252,E2 9446.252} C_VEL
LIN {X 0,Y 238.103,Z 1106.097,A -85,B 0,C 180,E1 9442.335,E2 9442.335} C_VEL
LIN {X 0,Y 227.495,Z 1117.642,A -85,B 0,C 180,E1 9438.562,E2 9438.562} C_VEL
LIN {X 0,Y 217.171,Z 1128.593,A -85,B 0,C 180,E1 9434.212,E2 9434.212} C_VEL
LIN {X 0,Y 205.711,Z 1140.682,A -85,B 0,C 180,E1 9428.186,E2 9428.186} C_VEL
LIN {X 0,Y 196.844,Z 1150.084,A -85,B 0,C 180,E1 9422.111,E2 9422.111} C_VEL
LIN {X 0,Y 190.656,Z 1157.086,A -85,B 0,C 180,E1 9416.499,E2 9416.499} C_VEL
LIN {X 0,Y 185.867,Z 1163.079,A -85,B 0,C 180,E1 9410.596,E2 9410.596} C_VEL
LIN {X 0,Y 182.377,Z 1168.401,A -85,B 0,C 180,E1 9404.094,E2 9404.094} C_VEL
LIN {X 0,Y 180.107,Z 1173.588,A -85,B 0,C 180,E1 9395.853,E2 9395.853} C_VEL
LIN {X 0,Y 179.596,Z 1176.762,A -85,B 0,C 180,E1 9388.971,E2 9388.971} C_VEL
LIN {X 0,Y 179.825,Z 1178.974,A -85,B 0,C 180,E1 9382.631,E2 9382.631} C_VEL
LIN {X 0,Y 180.836,Z 1180.536,A -85,B 0,C 180,E1 9376.379,E2 9376.379} C_VEL
LIN {X 0,Y 182.963,Z 1181.52,A -85,B 0,C 180,E1 9369.754,E2 9369.754} C_VEL
LIN {X 0,Y 187.17,Z 1181.793,A -85,B 0,C 180,E1 9362.607,E2 9362.607} C_VEL
LIN {X 0,Y 195.766,Z 1181.056,A -85,B 0,C 180,E1 9353.843,E2 9353.843} C_VEL
LIN {X 0,Y 209.524,Z 1178.497,A -85,B 0,C 180,E1 9345.066,E2 9345.066} C_VEL
LIN {X 0,Y 229.807,Z 1174.121,A -85,B 0,C 180,E1 9336.675,E2 9336.675} C_VEL
LIN {X 0,Y 242.317,Z 1171.302,A -85,B 0,C 180,E1 9332.84,E2 9332.84} C_VEL
LIN {X 0,Y 213.681,Z 1191.521,A -85,B 0,C 180,E1 9323.145,E2 9323.145} C_VEL
LIN {X 0,Y 199.671,Z 1203.175,A -85,B 0,C 180,E1 9315.732,E2 9315.732} C_VEL
LIN {X 0,Y 190.302,Z 1212.325,A -85,B 0,C 180,E1 9308.475,E2 9308.475} C_VEL
LIN {X 0,Y 184.257,Z 1219.543,A -85,B 0,C 180,E1 9301.396,E2 9301.396} C_VEL
LIN {X 0,Y 180.744,Z 1225.224,A -85,B 0,C 180,E1 9294.513,E2 9294.513} C_VEL
LIN {X 0,Y 180.659,Z 1225.389,A -85,B 0,C 180,E1 9294.288,E2 9294.288} C_VEL
LIN {X 0,Y 178.907,Z 1227.048,A -85,B 0,C 180,E1 9291.93,E2 9291.93} C_VEL
LIN {X 0,Y 171.464,Z 1230.227,A -85,B 0,C 180,E1 9285.082,E2 9285.082} C_VEL
LIN {X 0,Y 170.941,Z 1230.872,A -85,B 0,C 180,E1 9283.234,E2 9283.234} C_VEL
LIN {X 0,Y 171.364,Z 1232.963,A -85,B 0,C 180,E1 9277.038,E2 9277.038} C_VEL
LIN {X 0,Y 171.868,Z 1233.835,A -85,B 0,C 180,E1 9272,E2 9272} C_VEL
LIN {X 0,Y 171.838,Z 1233.738,A -85,B 0,C 180,E1 9267.332,E2 9267.332} C_VEL
LIN {X 0,Y 171.398,Z 1232.974,A -85,B 0,C 180,E1 9262.963,E2 9262.963} C_VEL
LIN {X 0,Y 171.039,Z 1231.042,A -85,B 0,C 180,E1 9257.165,E2 9257.165} C_VEL
LIN {X 0,Y 171.553,Z 1227.661,A -85,B 0,C 180,E1 9250.596,E2 9250.596} C_VEL
LIN {X 0,Y 173.547,Z 1223.038,A -85,B 0,C 180,E1 9244,E2 9244} C_VEL
LIN {X 0,Y 177.155,Z 1217.238,A -85,B 0,C 180,E1 9237.575,E2 9237.575} C_VEL
LIN {X 0,Y 182.52,Z 1210.175,A -85,B 0,C 180,E1 9231.354,E2 9231.354} C_VEL
LIN {X 0,Y 189.818,Z 1201.623,A -85,B 0,C 180,E1 9225.327,E2 9225.327} C_VEL
LIN {X 0,Y 200.901,Z 1189.4,A -85,B 0,C 180,E1 9218.613,E2 9218.613} C_VEL
LIN {X 0,Y 212.133,Z 1177.18,A -85,B 0,C 180,E1 9213.459,E2 9213.459} C_VEL
LIN {X 0,Y 222.808,Z 1165.452,A -85,B 0,C 180,E1 9209.472,E2 9209.472} C_VEL
LIN {X 0,Y 235.823,Z 1150.766,A -85,B 0,C 180,E1 9205.43,E2 9205.43} C_VEL
LIN {X 0,Y 251.375,Z 1132.262,A -85,B 0,C 180,E1 9201.446,E2 9201.446} C_VEL
LIN {X 0,Y 264.345,Z 1115.891,A -85,B 0,C 180,E1 9198.647,E2 9198.647} C_VEL
LIN {X 0,Y 277.634,Z 1098.112,A -85,B 0,C 180,E1 9196.159,E2 9196.159} C_VEL
LIN {X 0,Y 293.605,Z 1074.886,A -85,B 0,C 180,E1 9193.565,E2 9193.565} C_VEL
LIN {X 0,Y 305.948,Z 1055.342,A -85,B 0,C 180,E1 9191.818,E2 9191.818} C_VEL
LIN {X 0,Y 318.966,Z 1032.953,A -85,B 0,C 180,E1 9190.163,E2 9190.163} C_VEL
LIN {X 0,Y 331.795,Z 1008.361,A -85,B 0,C 180,E1 9188.721,E2 9188.721} C_VEL
LIN {X 0,Y 342.031,Z 986.638,A -85,B 0,C 180,E1 9187.686,E2 9187.686} C_VEL
LIN {X 0,Y 352.998,Z 960.801,A -85,B 0,C 180,E1 9186.69,E2 9186.69} C_VEL
LIN {X 0,Y 362.63,Z 934.306,A -85,B 0,C 180,E1 9185.907,E2 9185.907} C_VEL
LIN {X 0,Y 369.819,Z 911.54,A -85,B 0,C 180,E1 9185.357,E2 9185.357} C_VEL
LIN {X 0,Y 377.161,Z 883.331,A -85,B 0,C 180,E1 9184.743,E2 9184.743} C_VEL
LIN {X 0,Y 382.539,Z 855.89,A -85,B 0,C 180,E1 9184.233,E2 9184.233} C_VEL
LIN {X 0,Y 410.636,Z 672.353,A -85,B 0,C 180,E1 9181.36,E2 9181.36} C_VEL
LIN {X 0,Y 405.192,Z 662.541,A -85,B 0,C 180,E1 9178.016,E2 9178.016} C_VEL
LIN {X 0,Y 399.43,Z 652.526,A -85,B 0,C 180,E1 9173.893,E2 9173.893} C_VEL
LIN {X 0,Y 394.46,Z 644.311,A -85,B 0,C 180,E1 9169.779,E2 9169.779} C_VEL
LIN {X 0,Y 390.8,Z 638.522,A -85,B 0,C 180,E1 9166.159,E2 9166.159} C_VEL
LIN {X 0,Y 388.415,Z 634.366,A -85,B 0,C 180,E1 9163.243,E2 9163.243} C_VEL
LIN {X 0,Y 386.388,Z 631.294,A -85,B 0,C 180,E1 9160.38,E2 9160.38} C_VEL
LIN {X 0,Y 383.517,Z 628.293,A -85,B 0,C 180,E1 9155.674,E2 9155.674} C_VEL
LIN {X 0,Y 382.449,Z 625.867,A -85,B 0,C 180,E1 9152.604,E2 9152.604} C_VEL
LIN {X 0,Y 381.215,Z 625.235,A -85,B 0,C 180,E1 9147.907,E2 9147.907} C_VEL
LIN {X 0,Y 381.014,Z 625.078,A -85,B 0,C 180,E1 9142.873,E2 9142.873} C_VEL
LIN {X 0,Y 381.954,Z 625.493,A -85,B 0,C 180,E1 9138.251,E2 9138.251} C_VEL
LIN {X 0,Y 383.12,Z 626.234,A -85,B 0,C 180,E1 9135.197,E2 9135.197} C_VEL
LIN {X 0,Y 385.682,Z 630.261,A -85,B 0,C 180,E1 9130.205,E2 9130.205} C_VEL
LIN {X 0,Y 387.693,Z 632.092,A -85,B 0,C 180,E1 9127.595,E2 9127.595} C_VEL
LIN {X 0,Y 391.366,Z 636.754,A -85,B 0,C 180,E1 9123.494,E2 9123.494} C_VEL
LIN {X 0,Y 395.859,Z 642.917,A -85,B 0,C 180,E1 9119.453,E2 9119.453} C_VEL
LIN {X 0,Y 399.65,Z 648.051,A -85,B 0,C 180,E1 9116.605,E2 9116.605} C_VEL
LIN {X 0,Y 404.892,Z 655.363,A -85,B 0,C 180,E1 9113.175,E2 9113.175} C_VEL
LIN {X 0,Y 406.824,Z 658.391,A -85,B 0,C 180,E1 9112.001,E2 9112.001} C_VEL
LIN {X 0,Y 384.262,Z 805.921,A -85,B 0,C 180,E1 9109.728,E2 9109.728} C_VEL
LIN {X 0,Y 377.931,Z 836.855,A -85,B 0,C 180,E1 9109.07,E2 9109.07} C_VEL
LIN {X 0,Y 371.876,Z 860.64,A -85,B 0,C 180,E1 9108.425,E2 9108.425} C_VEL
LIN {X 0,Y 363.697,Z 887.878,A -85,B 0,C 180,E1 9107.528,E2 9107.528} C_VEL
LIN {X 0,Y 354.199,Z 914.196,A -85,B 0,C 180,E1 9106.455,E2 9106.455} C_VEL
LIN {X 0,Y 345.146,Z 936.411,A -85,B 0,C 180,E1 9105.371,E2 9105.371} C_VEL
LIN {X 0,Y 333.186,Z 962.368,A -85,B 0,C 180,E1 9103.854,E2 9103.854} C_VEL
LIN {X 0,Y 322.188,Z 983.49,A -85,B 0,C 180,E1 9102.365,E2 9102.365} C_VEL
LIN {X 0,Y 311.048,Z 1003.025,A -85,B 0,C 180,E1 9100.745,E2 9100.745} C_VEL
LIN {X 0,Y 297.088,Z 1025.405,A -85,B 0,C 180,E1 9098.516,E2 9098.516} C_VEL
LIN {X 0,Y 283.592,Z 1044.889,A -85,B 0,C 180,E1 9096.128,E2 9096.128} C_VEL
LIN {X 0,Y 271.277,Z 1061.39,A -85,B 0,C 180,E1 9093.698,E2 9093.698} C_VEL
LIN {X 0,Y 256.506,Z 1079.898,A -85,B 0,C 180,E1 9090.372,E2 9090.372} C_VEL
LIN {X 0,Y 242.868,Z 1095.592,A -85,B 0,C 180,E1 9086.829,E2 9086.829} C_VEL
LIN {X 0,Y 231.218,Z 1108.388,A -85,B 0,C 180,E1 9083.295,E2 9083.295} C_VEL
LIN {X 0,Y 219.825,Z 1120.41,A -85,B 0,C 180,E1 9079.252,E2 9079.252} C_VEL
LIN {X 0,Y 206.409,Z 1134.142,A -85,B 0,C 180,E1 9073.393,E2 9073.393} C_VEL
LIN {X 0,Y 196.486,Z 1144.145,A -85,B 0,C 180,E1 9067.879,E2 9067.879} C_VEL
LIN {X 0,Y 189.021,Z 1151.89,A -85,B 0,C 180,E1 9062.6,E2 9062.6} C_VEL
LIN {X 0,Y 182.741,Z 1158.791,A -85,B 0,C 180,E1 9056.828,E2 9056.828} C_VEL
LIN {X 0,Y 177.186,Z 1165.707,A -85,B 0,C 180,E1 9049.626,E2 9049.626} C_VEL
LIN {X 0,Y 173.356,Z 1171.856,A -85,B 0,C 180,E1 9041.112,E2 9041.112} C_VEL
LIN {X 0,Y 172.002,Z 1175.594,A -85,B 0,C 180,E1 9034.325,E2 9034.325} C_VEL
LIN {X 0,Y 171.663,Z 1178.203,A -85,B 0,C 180,E1 9028.416,E2 9028.416} C_VEL
LIN {X 0,Y 171.966,Z 1180.366,A -85,B 0,C 180,E1 9022.206,E2 9022.206} C_VEL
LIN {X 0,Y 173.175,Z 1182.075,A -85,B 0,C 180,E1 9015.374,E2 9015.374} C_VEL
LIN {X 0,Y 175.748,Z 1183.19,A -85,B 0,C 180,E1 9008.177,E2 9008.177} C_VEL
LIN {X 0,Y 180.417,Z 1183.551,A -85,B 0,C 180,E1 9000.953,E2 9000.953} C_VEL
LIN {X 0,Y 190.09,Z 1182.959,A -85,B 0,C 180,E1 8991.835,E2 8991.835} C_VEL
LIN {X 0,Y 205.025,Z 1180.618,A -85,B 0,C 180,E1 8982.985,E2 8982.985} C_VEL
LIN {X 0,Y 227.284,Z 1176.471,A -85,B 0,C 180,E1 8974.461,E2 8974.461} C_VEL
LIN {X 0,Y 232.105,Z 1175.556,A -85,B 0,C 180,E1 8972.955,E2 8972.955} C_VEL
LIN {X 0,Y 205.753,Z 1193.187,A -85,B 0,C 180,E1 8963.774,E2 8963.774} C_VEL
LIN {X 0,Y 187.647,Z 1207.616,A -85,B 0,C 180,E1 8953.422,E2 8953.422} C_VEL
LIN {X 0,Y 178.844,Z 1216.269,A -85,B 0,C 180,E1 8945.159,E2 8945.159} C_VEL
LIN {X 0,Y 173.873,Z 1222.722,A -85,B 0,C 180,E1 8937.39,E2 8937.39} C_VEL
LIN {X 0,Y 171.518,Z 1227.474,A -85,B 0,C 180,E1 8930.117,E2 8930.117} C_VEL
LIN {X 0,Y 170.941,Z 1230.872,A -85,B 0,C 180,E1 8923.234,E2 8923.234} C_VEL
LIN {X 0,Y 170.235,Z 1231.659,A -85,B 0,C 180,E1 8920.839,E2 8920.839} C_VEL
LIN {X 0,Y 167.688,Z 1232.245,A -85,B 0,C 180,E1 8917.545,E2 8917.545} C_VEL
LIN {X 0,Y 164.187,Z 1232.462,A -85,B 0,C 180,E1 8912.397,E2 8912.397} C_VEL
LIN {X 0,Y 164.023,Z 1232.438,A -85,B 0,C 180,E1 8911.212,E2 8911.212} C_VEL
LIN {X 0,Y 163.902,Z 1232.221,A -85,B 0,C 180,E1 8906.502,E2 8906.502} C_VEL
LIN {X 0,Y 163.299,Z 1230.82,A -85,B 0,C 180,E1 8900.338,E2 8900.338} C_VEL
LIN {X 0,Y 163.348,Z 1227.728,A -85,B 0,C 180,E1 8892.73,E2 8892.73} C_VEL
LIN {X 0,Y 165.605,Z 1222.099,A -85,B 0,C 180,E1 8883.848,E2 8883.848} C_VEL
LIN {X 0,Y 169.588,Z 1216.007,A -85,B 0,C 180,E1 8876.748,E2 8876.748} C_VEL
LIN {X 0,Y 175.247,Z 1208.944,A -85,B 0,C 180,E1 8870.281,E2 8870.281} C_VEL
LIN {X 0,Y 182.722,Z 1200.603,A -85,B 0,C 180,E1 8864.205,E2 8864.205} C_VEL
LIN {X 0,Y 193.982,Z 1188.727,A -85,B 0,C 180,E1 8857.459,E2 8857.459} C_VEL
LIN {X 0,Y 206.22,Z 1175.883,A -85,B 0,C 180,E1 8851.951,E2 8851.951} C_VEL
LIN {X 0,Y 217.286,Z 1164.138,A -85,B 0,C 180,E1 8847.93,E2 8847.93} C_VEL
LIN {X 0,Y 229.992,Z 1150.244,A -85,B 0,C 180,E1 8844.082,E2 8844.082} C_VEL
LIN {X 0,Y 246.316,Z 1131.393,A -85,B 0,C 180,E1 8840.005,E2 8840.005} C_VEL
LIN {X 0,Y 260.02,Z 1114.507,A -85,B 0,C 180,E1 8837.142,E2 8837.142} C_VEL
LIN {X 0,Y 273.867,Z 1096.363,A -85,B 0,C 180,E1 8834.647,E2 8834.647} C_VEL
LIN {X 0,Y 289.905,Z 1073.422,A -85,B 0,C 180,E1 8832.145,E2 8832.145} C_VEL
LIN {X 0,Y 302.468,Z 1053.856,A -85,B 0,C 180,E1 8830.438,E2 8830.438} C_VEL
LIN {X 0,Y 316.062,Z 1030.817,A -85,B 0,C 180,E1 8828.785,E2 8828.785} C_VEL
LIN {X 0,Y 328.715,Z 1006.755,A -85,B 0,C 180,E1 8827.424,E2 8827.424} C_VEL
LIN {X 0,Y 339.086,Z 984.988,A -85,B 0,C 180,E1 8826.423,E2 8826.423} C_VEL
LIN {X 0,Y 350.051,Z 959.398,A -85,B 0,C 180,E1 8825.471,E2 8825.471} C_VEL
LIN {X 0,Y 359.918,Z 932.507,A -85,B 0,C 180,E1 8824.706,E2 8824.706} C_VEL
LIN {X 0,Y 367.662,Z 908.03,A -85,B 0,C 180,E1 8824.137,E2 8824.137} C_VEL
LIN {X 0,Y 375.38,Z 877.445,A -85,B 0,C 180,E1 8823.503,E2 8823.503} C_VEL
LIN {X 0,Y 380.243,Z 852.348,A -85,B 0,C 180,E1 8823.051,E2 8823.051} C_VEL
LIN {X 0,Y 407.428,Z 677.589,A -85,B 0,C 180,E1 8820.352,E2 8820.352} C_VEL
LIN {X 0,Y 401.935,Z 667.829,A -85,B 0,C 180,E1 8816.863,E2 8816.863} C_VEL
LIN {X 0,Y 397.004,Z 659.358,A -85,B 0,C 180,E1 8813.274,E2 8813.274} C_VEL
LIN {X 0,Y 392.545,Z 651.838,A -85,B 0,C 180,E1 8809.484,E2 8809.484} C_VEL
LIN {X 0,Y 388.953,Z 646.077,A -85,B 0,C 180,E1 8805.864,E2 8805.864} C_VEL
LIN {X 0,Y 386.646,Z 642.028,A -85,B 0,C 180,E1 8803.009,E2 8803.009} C_VEL
LIN {X 0,Y 384.72,Z 639.085,A -85,B 0,C 180,E1 8800.253,E2 8800.253} C_VEL
LIN {X 0,Y 381.901,Z 636.094,A -85,B 0,C 180,E1 8795.564,E2 8795.564} C_VEL
LIN {X 0,Y 380.835,Z 633.692,A -85,B 0,C 180,E1 8792.478,E2 8792.478} C_VEL
LIN {X 0,Y 379.629,Z 633.02,A -85,B 0,C 180,E1 8787.439,E2 8787.439} C_VEL
LIN {X 0,Y 379.469,Z 632.935,A -85,B 0,C 180,E1 8782.696,E2 8782.696} C_VEL
LIN {X 0,Y 380.527,Z 633.387,A -85,B 0,C 180,E1 8777.929,E2 8777.929} C_VEL
LIN {X 0,Y 381.548,Z 634.109,A -85,B 0,C 180,E1 8775.249,E2 8775.249} C_VEL
LIN {X 0,Y 384.155,Z 638.14,A -85,B 0,C 180,E1 8770.203,E2 8770.203} C_VEL
LIN {X 0,Y 386.087,Z 639.956,A -85,B 0,C 180,E1 8767.675,E2 8767.675} C_VEL
LIN {X 0,Y 390.237,Z 645.388,A -85,B 0,C 180,E1 8763.076,E2 8763.076} C_VEL
LIN {X 0,Y 394.094,Z 650.605,A -85,B 0,C 180,E1 8759.653,E2 8759.653} C_VEL
LIN {X 0,Y 397.892,Z 655.784,A -85,B 0,C 180,E1 8756.783,E2 8756.783} C_VEL
LIN {X 0,Y 403.049,Z 663.069,A -85,B 0,C 180,E1 8753.378,E2 8753.378} C_VEL
LIN {X 0,Y 403.602,Z 664.229,A -85,B 0,C 180,E1 8753,E2 8753} C_VEL
LIN {X 0,Y 381.447,Z 806.584,A -85,B 0,C 180,E1 8750.845,E2 8750.845} C_VEL
LIN {X 0,Y 374.998,Z 837.682,A -85,B 0,C 180,E1 8750.197,E2 8750.197} C_VEL
LIN {X 0,Y 368.574,Z 862.46,A -85,B 0,C 180,E1 8749.535,E2 8749.535} C_VEL
LIN {X 0,Y 359.999,Z 890.285,A -85,B 0,C 180,E1 8748.627,E2 8748.627} C_VEL
LIN {X 0,Y 350.59,Z 915.883,A -85,B 0,C 180,E1 8747.596,E2 8747.596} C_VEL
LIN {X 0,Y 340.976,Z 939.013,A -85,B 0,C 180,E1 8746.482,E2 8746.482} C_VEL
LIN {X 0,Y 328.175,Z 965.965,A -85,B 0,C 180,E1 8744.905,E2 8744.905} C_VEL
LIN {X 0,Y 317.411,Z 986.174,A -85,B 0,C 180,E1 8743.48,E2 8743.48} C_VEL
LIN {X 0,Y 304.808,Z 1007.761,A -85,B 0,C 180,E1 8741.679,E2 8741.679} C_VEL
LIN {X 0,Y 290.391,Z 1029.906,A -85,B 0,C 180,E1 8739.417,E2 8739.417} C_VEL
LIN {X 0,Y 278.228,Z 1047.042,A -85,B 0,C 180,E1 8737.302,E2 8737.302} C_VEL
LIN {X 0,Y 265.638,Z 1063.549,A -85,B 0,C 180,E1 8734.869,E2 8734.869} C_VEL
LIN {X 0,Y 249.545,Z 1083.075,A -85,B 0,C 180,E1 8731.301,E2 8731.301} C_VEL
LIN {X 0,Y 236.631,Z 1097.573,A -85,B 0,C 180,E1 8727.983,E2 8727.983} C_VEL
LIN {X 0,Y 224.585,Z 1110.439,A -85,B 0,C 180,E1 8724.379,E2 8724.379} C_VEL
LIN {X 0,Y 211.284,Z 1124.099,A -85,B 0,C 180,E1 8719.64,E2 8719.64} C_VEL
LIN {X 0,Y 198.37,Z 1136.739,A -85,B 0,C 180,E1 8713.905,E2 8713.905} C_VEL
LIN {X 0,Y 188.855,Z 1146.032,A -85,B 0,C 180,E1 8708.573,E2 8708.573} C_VEL
LIN {X 0,Y 180.614,Z 1154.308,A -85,B 0,C 180,E1 8702.646,E2 8702.646} C_VEL
LIN {X 0,Y 172.581,Z 1163.083,A -85,B 0,C 180,E1 8694.594,E2 8694.594} C_VEL
LIN {X 0,Y 167.795,Z 1169.208,A -85,B 0,C 180,E1 8687.135,E2 8687.135} C_VEL
LIN {X 0,Y 165.176,Z 1173.68,A -85,B 0,C 180,E1 8680.295,E2 8680.295} C_VEL
LIN {X 0,Y 164.026,Z 1177.145,A -85,B 0,C 180,E1 8673.692,E2 8673.692} C_VEL
LIN {X 0,Y 163.749,Z 1179.719,A -85,B 0,C 180,E1 8667.65,E2 8667.65} C_VEL
LIN {X 0,Y 164.208,Z 1181.924,A -85,B 0,C 180,E1 8661.055,E2 8661.055} C_VEL
LIN {X 0,Y 165.631,Z 1183.691,A -85,B 0,C 180,E1 8653.974,E2 8653.974} C_VEL
LIN {X 0,Y 168.686,Z 1184.874,A -85,B 0,C 180,E1 8646.467,E2 8646.467} C_VEL
LIN {X 0,Y 174.008,Z 1185.339,A -85,B 0,C 180,E1 8638.934,E2 8638.934} C_VEL
LIN {X 0,Y 185.144,Z 1184.857,A -85,B 0,C 180,E1 8629.386,E2 8629.386} C_VEL
LIN {X 0,Y 202.505,Z 1182.573,A -85,B 0,C 180,E1 8620.081,E2 8620.081} C_VEL
LIN {X 0,Y 222.006,Z 1179.562,A -85,B 0,C 180,E1 8613.095,E2 8613.095} C_VEL
LIN {X 0,Y 193.856,Z 1197.419,A -85,B 0,C 180,E1 8602.59,E2 8602.59} C_VEL
LIN {X 0,Y 180.1,Z 1207.807,A -85,B 0,C 180,E1 8594.259,E2 8594.259} C_VEL
LIN {X 0,Y 171.645,Z 1215.436,A -85,B 0,C 180,E1 8586.454,E2 8586.454} C_VEL
LIN {X 0,Y 166.622,Z 1221.219,A -85,B 0,C 180,E1 8579.082,E2 8579.082} C_VEL
LIN {X 0,Y 163.917,Z 1225.748,A -85,B 0,C 180,E1 8571.845,E2 8571.845} C_VEL
LIN {X 0,Y 163.022,Z 1229.231,A -85,B 0,C 180,E1 8564.564,E2 8564.564} C_VEL
LIN {X 0,Y 163.351,Z 1231.384,A -85,B 0,C 180,E1 8558.093,E2 8558.093} C_VEL
LIN {X 0,Y 163.935,Z 1232.352,A -85,B 0,C 180,E1 8552.797,E2 8552.797} C_VEL
LIN {X 0,Y 164.023,Z 1232.438,A -85,B 0,C 180,E1 8551.212,E2 8551.212} C_VEL
LIN {X 0,Y 163.236,Z 1232.226,A -85,B 0,C 180,E1 8548.906,E2 8548.906} C_VEL
LIN {X 0,Y 160.378,Z 1231.528,A -85,B 0,C 180,E1 8545.708,E2 8545.708} C_VEL
LIN {X 0,Y 155.661,Z 1229.544,A -85,B 0,C 180,E1 8540.227,E2 8540.227} C_VEL
LIN {X 0,Y 155.312,Z 1228.978,A -85,B 0,C 180,E1 8538.781,E2 8538.781} C_VEL
LIN {X 0,Y 155.732,Z 1225.294,A -85,B 0,C 180,E1 8530.496,E2 8530.496} C_VEL
LIN {X 0,Y 157.999,Z 1220.515,A -85,B 0,C 180,E1 8522.894,E2 8522.894} C_VEL
LIN {X 0,Y 162.063,Z 1214.715,A -85,B 0,C 180,E1 8515.844,E2 8515.844} C_VEL
LIN {X 0,Y 168.044,Z 1207.661,A -85,B 0,C 180,E1 8509.118,E2 8509.118} C_VEL
LIN {X 0,Y 175.919,Z 1199.327,A -85,B 0,C 180,E1 8502.844,E2 8502.844} C_VEL
LIN {X 0,Y 188.285,Z 1186.847,A -85,B 0,C 180,E1 8495.659,E2 8495.659} C_VEL
LIN {X 0,Y 200.455,Z 1174.585,A -85,B 0,C 180,E1 8490.353,E2 8490.353} C_VEL
LIN {X 0,Y 212.628,Z 1162.101,A -85,B 0,C 180,E1 8486.081,E2 8486.081} C_VEL
LIN {X 0,Y 228.079,Z 1145.666,A -85,B 0,C 180,E1 8481.661,E2 8481.661} C_VEL
LIN {X 0,Y 243.47,Z 1128.065,A -85,B 0,C 180,E1 8478.062,E2 8478.062} C_VEL
LIN {X 0,Y 256.302,Z 1112.532,A -85,B 0,C 180,E1 8475.51,E2 8475.51} C_VEL
LIN {X 0,Y 272.159,Z 1092.038,A -85,B 0,C 180,E1 8472.794,E2 8472.794} C_VEL
LIN {X 0,Y 286.88,Z 1071.05,A -85,B 0,C 180,E1 8470.621,E2 8470.621} C_VEL
LIN {X 0,Y 299.626,Z 1051.411,A -85,B 0,C 180,E1 8468.968,E2 8468.968} C_VEL
LIN {X 0,Y 313.912,Z 1027.281,A -85,B 0,C 180,E1 8467.32,E2 8467.32} C_VEL
LIN {X 0,Y 325.806,Z 1004.82,A -85,B 0,C 180,E1 8466.103,E2 8466.103} C_VEL
LIN {X 0,Y 336.31,Z 982.985,A -85,B 0,C 180,E1 8465.138,E2 8465.138} C_VEL
LIN {X 0,Y 347.884,Z 955.93,A -85,B 0,C 180,E1 8464.184,E2 8464.184} C_VEL
LIN {X 0,Y 357.123,Z 930.901,A -85,B 0,C 180,E1 8463.505,E2 8463.505} C_VEL
LIN {X 0,Y 364.891,Z 906.542,A -85,B 0,C 180,E1 8462.958,E2 8462.958} C_VEL
LIN {X 0,Y 372.529,Z 876.546,A -85,B 0,C 180,E1 8462.352,E2 8462.352} C_VEL
LIN {X 0,Y 377.365,Z 852.006,A -85,B 0,C 180,E1 8461.918,E2 8461.918} C_VEL
LIN {X 0,Y 404.126,Z 682.955,A -85,B 0,C 180,E1 8459.362,E2 8459.362} C_VEL
LIN {X 0,Y 399.655,Z 674.912,A -85,B 0,C 180,E1 8456.414,E2 8456.414} C_VEL
LIN {X 0,Y 395.092,Z 666.929,A -85,B 0,C 180,E1 8453.023,E2 8453.023} C_VEL
LIN {X 0,Y 390.872,Z 659.687,A -85,B 0,C 180,E1 8449.386,E2 8449.386} C_VEL
LIN {X 0,Y 387.138,Z 653.66,A -85,B 0,C 180,E1 8445.587,E2 8445.587} C_VEL
LIN {X 0,Y 384.884,Z 649.69,A -85,B 0,C 180,E1 8442.773,E2 8442.773} C_VEL
LIN {X 0,Y 383.087,Z 646.897,A -85,B 0,C 180,E1 8440.165,E2 8440.165} C_VEL
LIN {X 0,Y 380.357,Z 644.017,A -85,B 0,C 180,E1 8435.624,E2 8435.624} C_VEL
LIN {X 0,Y 379.222,Z 641.519,A -85,B 0,C 180,E1 8432.351,E2 8432.351} C_VEL
LIN {X 0,Y 378.037,Z 640.842,A -85,B 0,C 180,E1 8427.255,E2 8427.255} C_VEL
LIN {X 0,Y 377.928,Z 640.787,A -85,B 0,C 180,E1 8422.517,E2 8422.517} C_VEL
LIN {X 0,Y 379.135,Z 641.328,A -85,B 0,C 180,E1 8417.534,E2 8417.534} C_VEL
LIN {X 0,Y 379.957,Z 641.923,A -85,B 0,C 180,E1 8415.361,E2 8415.361} C_VEL
LIN {X 0,Y 382.59,Z 645.98,A -85,B 0,C 180,E1 8410.258,E2 8410.258} C_VEL
LIN {X 0,Y 384.398,Z 647.666,A -85,B 0,C 180,E1 8407.87,E2 8407.87} C_VEL
LIN {X 0,Y 388.551,Z 653.145,A -85,B 0,C 180,E1 8403.238,E2 8403.238} C_VEL
LIN {X 0,Y 392.298,Z 658.235,A -85,B 0,C 180,E1 8399.887,E2 8399.887} C_VEL
LIN {X 0,Y 396.102,Z 663.463,A -85,B 0,C 180,E1 8396.989,E2 8396.989} C_VEL
LIN {X 0,Y 400.514,Z 669.823,A -85,B 0,C 180,E1 8394.017,E2 8394.017} C_VEL
LIN {X 0,Y 378.676,Z 807.595,A -85,B 0,C 180,E1 8391.97,E2 8391.97} C_VEL
LIN {X 0,Y 372.127,Z 838.644,A -85,B 0,C 180,E1 8391.336,E2 8391.336} C_VEL
LIN {X 0,Y 365.872,Z 862.51,A -85,B 0,C 180,E1 8390.713,E2 8390.713} C_VEL
LIN {X 0,Y 357.474,Z 889.726,A -85,B 0,C 180,E1 8389.854,E2 8389.854} C_VEL
LIN {X 0,Y 347.861,Z 915.682,A -85,B 0,C 180,E1 8388.841,E2 8388.841} C_VEL
LIN {X 0,Y 338.383,Z 938.321,A -85,B 0,C 180,E1 8387.782,E2 8387.782} C_VEL
LIN {X 0,Y 325.899,Z 964.584,A -85,B 0,C 180,E1 8386.304,E2 8386.304} C_VEL
LIN {X 0,Y 314.145,Z 986.417,A -85,B 0,C 180,E1 8384.812,E2 8384.812} C_VEL
LIN {X 0,Y 302.307,Z 1006.441,A -85,B 0,C 180,E1 8383.192,E2 8383.192} C_VEL
LIN {X 0,Y 286.568,Z 1030.439,A -85,B 0,C 180,E1 8380.814,E2 8380.814} C_VEL
LIN {X 0,Y 274.147,Z 1047.65,A -85,B 0,C 180,E1 8378.729,E2 8378.729} C_VEL
LIN {X 0,Y 261.48,Z 1063.963,A -85,B 0,C 180,E1 8376.367,E2 8376.367} C_VEL
LIN {X 0,Y 245.853,Z 1082.662,A -85,B 0,C 180,E1 8373.031,E2 8373.031} C_VEL
LIN {X 0,Y 231.982,Z 1097.893,A -85,B 0,C 180,E1 8369.605,E2 8369.605} C_VEL
LIN {X 0,Y 220.44,Z 1109.945,A -85,B 0,C 180,E1 8366.287,E2 8366.287} C_VEL
LIN {X 0,Y 209.355,Z 1121.024,A -85,B 0,C 180,E1 8362.591,E2 8362.591} C_VEL
LIN {X 0,Y 197.899,Z 1132.109,A -85,B 0,C 180,E1 8358.045,E2 8358.045} C_VEL
LIN {X 0,Y 184.624,Z 1144.709,A -85,B 0,C 180,E1 8351.366,E2 8351.366} C_VEL
LIN {X 0,Y 175.227,Z 1153.647,A -85,B 0,C 180,E1 8345.135,E2 8345.135} C_VEL
LIN {X 0,Y 168.153,Z 1160.781,A -85,B 0,C 180,E1 8338.901,E2 8338.901} C_VEL
LIN {X 0,Y 162.535,Z 1167.077,A -85,B 0,C 180,E1 8332.035,E2 8332.035} C_VEL
LIN {X 0,Y 158.241,Z 1173.228,A -85,B 0,C 180,E1 8323.531,E2 8323.531} C_VEL
LIN {X 0,Y 156.215,Z 1177.94,A -85,B 0,C 180,E1 8314.727,E2 8314.727} C_VEL
LIN {X 0,Y 155.842,Z 1180.971,A -85,B 0,C 180,E1 8307.514,E2 8307.514} C_VEL
LIN {X 0,Y 156.453,Z 1183.441,A -85,B 0,C 180,E1 8300.039,E2 8300.039} C_VEL
LIN {X 0,Y 158.184,Z 1185.315,A -85,B 0,C 180,E1 8292.411,E2 8292.411} C_VEL
LIN {X 0,Y 161.977,Z 1186.616,A -85,B 0,C 180,E1 8284.248,E2 8284.248} C_VEL
LIN {X 0,Y 168.698,Z 1187.18,A -85,B 0,C 180,E1 8275.921,E2 8275.921} C_VEL
LIN {X 0,Y 183.325,Z 1186.501,A -85,B 0,C 180,E1 8265.147,E2 8265.147} C_VEL
LIN {X 0,Y 204.362,Z 1184.241,A -85,B 0,C 180,E1 8255.733,E2 8255.733} C_VEL
LIN {X 0,Y 211.689,Z 1183.172,A -85,B 0,C 180,E1 8253.215,E2 8253.215} C_VEL
LIN {X 0,Y 185.334,Z 1199.118,A -85,B 0,C 180,E1 8242.983,E2 8242.983} C_VEL
LIN {X 0,Y 168.386,Z 1211.328,A -85,B 0,C 180,E1 8231.686,E2 8231.686} C_VEL
LIN {X 0,Y 160.638,Z 1218.47,A -85,B 0,C 180,E1 8222.787,E2 8222.787} C_VEL
LIN {X 0,Y 156.669,Z 1223.611,A -85,B 0,C 180,E1 8214.509,E2 8214.509} C_VEL
LIN {X 0,Y 155.179,Z 1227.484,A -85,B 0,C 180,E1 8206.244,E2 8206.244} C_VEL
LIN {X 0,Y 155.388,Z 1229.865,A -85,B 0,C 180,E1 8198.884,E2 8198.884} C_VEL
LIN {X 0,Y 156.043,Z 1230.943,A -85,B 0,C 180,E1 8192.938,E2 8192.938} C_VEL
LIN {X 0,Y 156.151,Z 1230.891,A -85,B 0,C 180,E1 8188.165,E2 8188.165} C_VEL
LIN {X 0,Y 155.728,Z 1230.249,A -85,B 0,C 180,E1 8183.733,E2 8183.733} C_VEL
LIN {X 0,Y 155.312,Z 1228.978,A -85,B 0,C 180,E1 8178.781,E2 8178.781} C_VEL
LIN {X 0,Y 154.406,Z 1227.814,A -85,B 0,C 180,E1 8176.178,E2 8176.178} C_VEL
LIN {X 0,Y 151.051,Z 1225.368,A -85,B 0,C 180,E1 8171.835,E2 8171.835} C_VEL
LIN {X 0,Y 148.774,Z 1222.559,A -85,B 0,C 180,E1 8167.523,E2 8167.523} C_VEL
LIN {X 0,Y 148.898,Z 1221.57,A -85,B 0,C 180,E1 8165.838,E2 8165.838} C_VEL
LIN {X 0,Y 153.488,Z 1214.787,A -85,B 0,C 180,E1 8156.377,E2 8156.377} C_VEL
LIN {X 0,Y 159.783,Z 1207.579,A -85,B 0,C 180,E1 8148.924,E2 8148.924} C_VEL
LIN {X 0,Y 167.849,Z 1199.353,A -85,B 0,C 180,E1 8142.311,E2 8142.311} C_VEL
LIN {X 0,Y 177.567,Z 1189.909,A -85,B 0,C 180,E1 8136.368,E2 8136.368} C_VEL
LIN {X 0,Y 191.546,Z 1176.505,A -85,B 0,C 180,E1 8129.942,E2 8129.942} C_VEL
LIN {X 0,Y 205.302,Z 1162.876,A -85,B 0,C 180,E1 8125.059,E2 8125.059} C_VEL
LIN {X 0,Y 217.975,Z 1149.865,A -85,B 0,C 180,E1 8121.38,E2 8121.38} C_VEL
LIN {X 0,Y 233.866,Z 1132.761,A -85,B 0,C 180,E1 8117.557,E2 8117.557} C_VEL
LIN {X 0,Y 249.843,Z 1114.04,A -85,B 0,C 180,E1 8114.367,E2 8114.367} C_VEL
LIN {X 0,Y 262.854,Z 1097.798,A -85,B 0,C 180,E1 8112.148,E2 8112.148} C_VEL
LIN {X 0,Y 278.089,Z 1077.356,A -85,B 0,C 180,E1 8109.879,E2 8109.879} C_VEL
LIN {X 0,Y 293.26,Z 1054.783,A -85,B 0,C 180,E1 8107.919,E2 8107.919} C_VEL
LIN {X 0,Y 305.437,Z 1034.997,A -85,B 0,C 180,E1 8106.519,E2 8106.519} C_VEL
LIN {X 0,Y 319.234,Z 1010.465,A -85,B 0,C 180,E1 8105.119,E2 8105.119} C_VEL
LIN {X 0,Y 331.36,Z 985.988,A -85,B 0,C 180,E1 8104.026,E2 8104.026} C_VEL
LIN {X 0,Y 341.494,Z 963.251,A -85,B 0,C 180,E1 8103.211,E2 8103.211} C_VEL
LIN {X 0,Y 353.012,Z 933.55,A -85,B 0,C 180,E1 8102.385,E2 8102.385} C_VEL
LIN {X 0,Y 360.648,Z 910.405,A -85,B 0,C 180,E1 8101.875,E2 8101.875} C_VEL
LIN {X 0,Y 367.929,Z 883.942,A -85,B 0,C 180,E1 8101.337,E2 8101.337} C_VEL
LIN {X 0,Y 374.057,Z 854.904,A -85,B 0,C 180,E1 8100.822,E2 8100.822} C_VEL
LIN {X 0,Y 400.939,Z 688.422,A -85,B 0,C 180,E1 8098.357,E2 8098.357} C_VEL
LIN {X 0,Y 397.509,Z 682.17,A -85,B 0,C 180,E1 8096.033,E2 8096.033} C_VEL
LIN {X 0,Y 393.287,Z 674.651,A -85,B 0,C 180,E1 8092.844,E2 8092.844} C_VEL
LIN {X 0,Y 389.332,Z 667.84,A -85,B 0,C 180,E1 8089.419,E2 8089.419} C_VEL
LIN {X 0,Y 385.433,Z 661.404,A -85,B 0,C 180,E1 8085.425,E2 8085.425} C_VEL
LIN {X 0,Y 383.128,Z 657.351,A -85,B 0,C 180,E1 8082.535,E2 8082.535} C_VEL
LIN {X 0,Y 381.455,Z 654.71,A -85,B 0,C 180,E1 8080.077,E2 8080.077} C_VEL
LIN {X 0,Y 378.78,Z 651.881,A -85,B 0,C 180,E1 8075.603,E2 8075.603} C_VEL
LIN {X 0,Y 377.676,Z 649.373,A -85,B 0,C 180,E1 8072.399,E2 8072.399} C_VEL
LIN {X 0,Y 376.492,Z 648.701,A -85,B 0,C 180,E1 8067.339,E2 8067.339} C_VEL
LIN {X 0,Y 376.368,Z 648.634,A -85,B 0,C 180,E1 8062.527,E2 8062.527} C_VEL
LIN {X 0,Y 377.541,Z 649.154,A -85,B 0,C 180,E1 8057.638,E2 8057.638} C_VEL
LIN {X 0,Y 378.344,Z 649.683,A -85,B 0,C 180,E1 8055.524,E2 8055.524} C_VEL
LIN {X 0,Y 380.828,Z 653.614,A -85,B 0,C 180,E1 8050.627,E2 8050.627} C_VEL
LIN {X 0,Y 382.713,Z 655.375,A -85,B 0,C 180,E1 8048.066,E2 8048.066} C_VEL
LIN {X 0,Y 386.868,Z 660.902,A -85,B 0,C 180,E1 8043.402,E2 8043.402} C_VEL
LIN {X 0,Y 390.557,Z 665.943,A -85,B 0,C 180,E1 8040.078,E2 8040.078} C_VEL
LIN {X 0,Y 394.359,Z 671.223,A -85,B 0,C 180,E1 8037.154,E2 8037.154} C_VEL
LIN {X 0,Y 397.344,Z 675.672,A -85,B 0,C 180,E1 8035.039,E2 8035.039} C_VEL
LIN {X 0,Y 375.919,Z 808.628,A -85,B 0,C 180,E1 8033.104,E2 8033.104} C_VEL
LIN {X 0,Y 369.265,Z 839.673,A -85,B 0,C 180,E1 8032.482,E2 8032.482} C_VEL
LIN {X 0,Y 362.68,Z 864.37,A -85,B 0,C 180,E1 8031.85,E2 8031.85} C_VEL
LIN {X 0,Y 353.975,Z 891.895,A -85,B 0,C 180,E1 8030.993,E2 8030.993} C_VEL
LIN {X 0,Y 344.227,Z 917.743,A -85,B 0,C 180,E1 8030,E2 8030} C_VEL
LIN {X 0,Y 334.22,Z 941.183,A -85,B 0,C 180,E1 8028.919,E2 8028.919} C_VEL
LIN {X 0,Y 321.528,Z 967.226,A -85,B 0,C 180,E1 8027.463,E2 8027.463} C_VEL
LIN {X 0,Y 310.055,Z 988.183,A -85,B 0,C 180,E1 8026.05,E2 8026.05} C_VEL
LIN {X 0,Y 297.233,Z 1009.496,A -85,B 0,C 180,E1 8024.342,E2 8024.342} C_VEL
LIN {X 0,Y 282.3,Z 1031.749,A -85,B 0,C 180,E1 8022.155,E2 8022.155} C_VEL
LIN {X 0,Y 269.358,Z 1049.358,A -85,B 0,C 180,E1 8020.048,E2 8020.048} C_VEL
LIN {X 0,Y 255.701,Z 1066.581,A -85,B 0,C 180,E1 8017.561,E2 8017.561} C_VEL
LIN {X 0,Y 239.083,Z 1085.803,A -85,B 0,C 180,E1 8014.077,E2 8014.077} C_VEL
LIN {X 0,Y 226.004,Z 1099.808,A -85,B 0,C 180,E1 8010.895,E2 8010.895} C_VEL
LIN {X 0,Y 213.221,Z 1112.762,A -85,B 0,C 180,E1 8007.266,E2 8007.266} C_VEL
LIN {X 0,Y 198.346,Z 1127.142,A -85,B 0,C 180,E1 8002.177,E2 8002.177} C_VEL
LIN {X 0,Y 185.11,Z 1139.266,A -85,B 0,C 180,E1 7996.481,E2 7996.481} C_VEL
LIN {X 0,Y 175.028,Z 1148.443,A -85,B 0,C 180,E1 7990.997,E2 7990.997} C_VEL
LIN {X 0,Y 165.985,Z 1156.854,A -85,B 0,C 180,E1 7984.636,E2 7984.636} C_VEL
LIN {X 0,Y 157.132,Z 1165.776,A -85,B 0,C 180,E1 7975.817,E2 7975.817} C_VEL
LIN {X 0,Y 152.091,Z 1171.792,A -85,B 0,C 180,E1 7967.889,E2 7967.889} C_VEL
LIN {X 0,Y 149.266,Z 1176.409,A -85,B 0,C 180,E1 7960.214,E2 7960.214} C_VEL
LIN {X 0,Y 148.136,Z 1179.853,A -85,B 0,C 180,E1 7953.143,E2 7953.143} C_VEL
LIN {X 0,Y 147.994,Z 1182.673,A -85,B 0,C 180,E1 7946.029,E2 7946.029} C_VEL
LIN {X 0,Y 148.751,Z 1185.031,A -85,B 0,C 180,E1 7938.6,E2 7938.6} C_VEL
LIN {X 0,Y 150.842,Z 1186.962,A -85,B 0,C 180,E1 7930.697,E2 7930.697} C_VEL
LIN {X 0,Y 155.523,Z 1188.394,A -85,B 0,C 180,E1 7921.842,E2 7921.842} C_VEL
LIN {X 0,Y 165.592,Z 1189.166,A -85,B 0,C 180,E1 7911.318,E2 7911.318} C_VEL
LIN {X 0,Y 182.66,Z 1188.309,A -85,B 0,C 180,E1 7900.826,E2 7900.826} C_VEL
LIN {X 0,Y 201.388,Z 1186.685,A -85,B 0,C 180,E1 7893.34,E2 7893.34} C_VEL
LIN {X 0,Y 175.133,Z 1201.541,A -85,B 0,C 180,E1 7882.521,E2 7882.521} C_VEL
LIN {X 0,Y 162.09,Z 1210.289,A -85,B 0,C 180,E1 7873.7,E2 7873.7} C_VEL
LIN {X 0,Y 153.853,Z 1216.997,A -85,B 0,C 180,E1 7864.883,E2 7864.883} C_VEL
LIN {X 0,Y 149.246,Z 1222.087,A -85,B 0,C 180,E1 7856.242,E2 7856.242} C_VEL
LIN {X 0,Y 147.385,Z 1225.713,A -85,B 0,C 180,E1 7848.184,E2 7848.184} C_VEL
LIN {X 0,Y 147.379,Z 1228.247,A -85,B 0,C 180,E1 7840.16,E2 7840.16} C_VEL
LIN {X 0,Y 148.123,Z 1229.438,A -85,B 0,C 180,E1 7833.483,E2 7833.483} C_VEL
LIN {X 0,Y 148.298,Z 1229.434,A -85,B 0,C 180,E1 7828.454,E2 7828.454} C_VEL
LIN {X 0,Y 147.858,Z 1228.766,A -85,B 0,C 180,E1 7823.769,E2 7823.769} C_VEL
LIN {X 0,Y 147.388,Z 1227.05,A -85,B 0,C 180,E1 7817.462,E2 7817.462} C_VEL
LIN {X 0,Y 147.929,Z 1223.759,A -85,B 0,C 180,E1 7809.835,E2 7809.835} C_VEL
LIN {X 0,Y 148.898,Z 1221.57,A -85,B 0,C 180,E1 7805.838,E2 7805.838} C_VEL
LIN {X 0,Y 148.951,Z 1219.695,A -85,B 0,C 180,E1 7802.942,E2 7802.942} C_VEL
LIN {X 0,Y 146.942,Z 1213.273,A -85,B 0,C 180,E1 7795.111,E2 7795.111} C_VEL
LIN {X 0,Y 147.971,Z 1211.135,A -85,B 0,C 180,E1 7792.674,E2 7792.674} C_VEL
LIN {X 0,Y 156.422,Z 1202.6,A -85,B 0,C 180,E1 7784.281,E2 7784.281} C_VEL
LIN {X 0,Y 167.992,Z 1191.682,A -85,B 0,C 180,E1 7776.527,E2 7776.527} C_VEL
LIN {X 0,Y 178.765,Z 1181.754,A -85,B 0,C 180,E1 7771.156,E2 7771.156} C_VEL
LIN {X 0,Y 190.836,Z 1170.479,A -85,B 0,C 180,E1 7766.37,E2 7766.37} C_VEL
LIN {X 0,Y 206.314,Z 1155.594,A -85,B 0,C 180,E1 7761.487,E2 7761.487} C_VEL
LIN {X 0,Y 222.225,Z 1139.172,A -85,B 0,C 180,E1 7757.471,E2 7757.471} C_VEL
LIN {X 0,Y 236.14,Z 1123.951,A -85,B 0,C 180,E1 7754.537,E2 7754.537} C_VEL
LIN {X 0,Y 252.585,Z 1104.761,A -85,B 0,C 180,E1 7751.607,E2 7751.607} C_VEL
LIN {X 0,Y 268.428,Z 1084.352,A -85,B 0,C 180,E1 7749.211,E2 7749.211} C_VEL
LIN {X 0,Y 281.837,Z 1065.636,A -85,B 0,C 180,E1 7747.439,E2 7747.439} C_VEL
LIN {X 0,Y 297.401,Z 1041.868,A -85,B 0,C 180,E1 7745.636,E2 7745.636} C_VEL
LIN {X 0,Y 310.344,Z 1019.828,A -85,B 0,C 180,E1 7744.322,E2 7744.322} C_VEL
LIN {X 0,Y 321.832,Z 998.346,A -85,B 0,C 180,E1 7743.28,E2 7743.28} C_VEL
LIN {X 0,Y 335.206,Z 970.181,A -85,B 0,C 180,E1 7742.202,E2 7742.202} C_VEL
LIN {X 0,Y 345.122,Z 946.279,A -85,B 0,C 180,E1 7741.494,E2 7741.494} C_VEL
LIN {X 0,Y 354.996,Z 919.169,A -85,B 0,C 180,E1 7740.863,E2 7740.863} C_VEL
LIN {X 0,Y 363.123,Z 891.505,A -85,B 0,C 180,E1 7740.312,E2 7740.312} C_VEL
LIN {X 0,Y 369.18,Z 866.132,A -85,B 0,C 180,E1 7739.848,E2 7739.848} C_VEL
LIN {X 0,Y 376.079,Z 827.591,A -85,B 0,C 180,E1 7739.241,E2 7739.241} C_VEL
LIN {X 0,Y 397.856,Z 693.719,A -85,B 0,C 180,E1 7737.299,E2 7737.299} C_VEL
LIN {X 0,Y 392.362,Z 683.913,A -85,B 0,C 180,E1 7733.341,E2 7733.341} C_VEL
LIN {X 0,Y 388.226,Z 676.727,A -85,B 0,C 180,E1 7729.838,E2 7729.838} C_VEL
LIN {X 0,Y 384.021,Z 669.597,A -85,B 0,C 180,E1 7725.598,E2 7725.598} C_VEL
LIN {X 0,Y 381.38,Z 665.011,A -85,B 0,C 180,E1 7722.294,E2 7722.294} C_VEL
LIN {X 0,Y 379.825,Z 662.522,A -85,B 0,C 180,E1 7719.987,E2 7719.987} C_VEL
LIN {X 0,Y 377.276,Z 659.855,A -85,B 0,C 180,E1 7715.739,E2 7715.739} C_VEL
LIN {X 0,Y 376.065,Z 657.2,A -85,B 0,C 180,E1 7712.271,E2 7712.271} C_VEL
LIN {X 0,Y 374.891,Z 656.524,A -85,B 0,C 180,E1 7707.155,E2 7707.155} C_VEL
LIN {X 0,Y 374.824,Z 656.482,A -85,B 0,C 180,E1 7702.398,E2 7702.398} C_VEL
LIN {X 0,Y 376.126,Z 657.076,A -85,B 0,C 180,E1 7697.321,E2 7697.321} C_VEL
LIN {X 0,Y 376.782,Z 657.608,A -85,B 0,C 180,E1 7695.525,E2 7695.525} C_VEL
LIN {X 0,Y 379.445,Z 661.643,A -85,B 0,C 180,E1 7690.398,E2 7690.398} C_VEL
LIN {X 0,Y 381.143,Z 663.313,A -85,B 0,C 180,E1 7688.092,E2 7688.092} C_VEL
LIN {X 0,Y 385.191,Z 668.661,A -85,B 0,C 180,E1 7683.564,E2 7683.564} C_VEL
LIN {X 0,Y 388.861,Z 673.718,A -85,B 0,C 180,E1 7680.234,E2 7680.234} C_VEL
LIN {X 0,Y 392.504,Z 678.862,A -85,B 0,C 180,E1 7677.375,E2 7677.375} C_VEL
LIN {X 0,Y 394.302,Z 681.575,A -85,B 0,C 180,E1 7676.076,E2 7676.076} C_VEL
LIN {X 0,Y 373.332,Z 809.506,A -85,B 0,C 180,E1 7674.256,E2 7674.256} C_VEL
LIN {X 0,Y 366.588,Z 840.553,A -85,B 0,C 180,E1 7673.65,E2 7673.65} C_VEL
LIN {X 0,Y 360.081,Z 864.657,A -85,B 0,C 180,E1 7673.05,E2 7673.05} C_VEL
LIN {X 0,Y 351.205,Z 892.477,A -85,B 0,C 180,E1 7672.209,E2 7672.209} C_VEL
LIN {X 0,Y 341.089,Z 918.938,A -85,B 0,C 180,E1 7671.218,E2 7671.218} C_VEL
LIN {X 0,Y 330.677,Z 942.955,A -85,B 0,C 180,E1 7670.135,E2 7670.135} C_VEL
LIN {X 0,Y 317.756,Z 968.956,A -85,B 0,C 180,E1 7668.707,E2 7668.707} C_VEL
LIN {X 0,Y 306.41,Z 989.357,A -85,B 0,C 180,E1 7667.358,E2 7667.358} C_VEL
LIN {X 0,Y 292.755,Z 1011.688,A -85,B 0,C 180,E1 7665.6,E2 7665.6} C_VEL
LIN {X 0,Y 278.045,Z 1033.117,A -85,B 0,C 180,E1 7663.518,E2 7663.518} C_VEL
LIN {X 0,Y 265.317,Z 1050.133,A -85,B 0,C 180,E1 7661.519,E2 7661.519} C_VEL
LIN {X 0,Y 251.746,Z 1066.952,A -85,B 0,C 180,E1 7659.141,E2 7659.141} C_VEL
LIN {X 0,Y 234.079,Z 1087.003,A -85,B 0,C 180,E1 7655.564,E2 7655.564} C_VEL
LIN {X 0,Y 221.192,Z 1100.498,A -85,B 0,C 180,E1 7652.528,E2 7652.528} C_VEL
LIN {X 0,Y 208.479,Z 1113.084,A -85,B 0,C 180,E1 7649.046,E2 7649.046} C_VEL
LIN {X 0,Y 195.112,Z 1125.679,A -85,B 0,C 180,E1 7644.707,E2 7644.707} C_VEL
LIN {X 0,Y 179.652,Z 1139.55,A -85,B 0,C 180,E1 7638.399,E2 7638.399} C_VEL
LIN {X 0,Y 168.954,Z 1148.923,A -85,B 0,C 180,E1 7632.789,E2 7632.789} C_VEL
LIN {X 0,Y 160.1,Z 1156.799,A -85,B 0,C 180,E1 7626.83,E2 7626.83} C_VEL
LIN {X 0,Y 152.446,Z 1163.994,A -85,B 0,C 180,E1 7619.973,E2 7619.973} C_VEL
LIN {X 0,Y 145.562,Z 1171.493,A -85,B 0,C 180,E1 7610.806,E2 7610.806} C_VEL
LIN {X 0,Y 141.476,Z 1177.422,A -85,B 0,C 180,E1 7600.868,E2 7600.868} C_VEL
LIN {X 0,Y 140.193,Z 1181.186,A -85,B 0,C 180,E1 7592.824,E2 7592.824} C_VEL
LIN {X 0,Y 140.104,Z 1184.055,A -85,B 0,C 180,E1 7585.354,E2 7585.354} C_VEL
LIN {X 0,Y 140.981,Z 1186.457,A -85,B 0,C 180,E1 7577.757,E2 7577.757} C_VEL
LIN {X 0,Y 143.607,Z 1188.631,A -85,B 0,C 180,E1 7568.811,E2 7568.811} C_VEL
LIN {X 0,Y 149.03,Z 1190.162,A -85,B 0,C 180,E1 7559.616,E2 7559.616} C_VEL
LIN {X 0,Y 160.711,Z 1191.11,A -85,B 0,C 180,E1 7548.516,E2 7548.516} C_VEL
LIN {X 0,Y 179.998,Z 1190.428,A -85,B 0,C 180,E1 7537.806,E2 7537.806} C_VEL
LIN {X 0,Y 191.085,Z 1189.67,A -85,B 0,C 180,E1 7533.479,E2 7533.479} C_VEL
LIN {X 0,Y 164.926,Z 1203.854,A -85,B 0,C 180,E1 7522.011,E2 7522.011} C_VEL
LIN {X 0,Y 149.936,Z 1213.505,A -85,B 0,C 180,E1 7510.305,E2 7510.305} C_VEL
LIN {X 0,Y 142.875,Z 1219.543,A -85,B 0,C 180,E1 7500.257,E2 7500.257} C_VEL
LIN {X 0,Y 139.815,Z 1223.714,A -85,B 0,C 180,E1 7490.951,E2 7490.951} C_VEL
LIN {X 0,Y 139.339,Z 1226.526,A -85,B 0,C 180,E1 7482.011,E2 7482.011} C_VEL
LIN {X 0,Y 140.125,Z 1227.89,A -85,B 0,C 180,E1 7474.502,E2 7474.502} C_VEL
LIN {X 0,Y 140.451,Z 1227.998,A -85,B 0,C 180,E1 7469.592,E2 7469.592} C_VEL
LIN {X 0,Y 140.145,Z 1227.541,A -85,B 0,C 180,E1 7465.088,E2 7465.088} C_VEL
LIN {X 0,Y 139.528,Z 1225.822,A -85,B 0,C 180,E1 7458.005,E2 7458.005} C_VEL
LIN {X 0,Y 139.995,Z 1222.609,A -85,B 0,C 180,E1 7449.951,E2 7449.951} C_VEL
LIN {X 0,Y 142.368,Z 1218.138,A -85,B 0,C 180,E1 7441.93,E2 7441.93} C_VEL
LIN {X 0,Y 146.906,Z 1212.352,A -85,B 0,C 180,E1 7434.092,E2 7434.092} C_VEL
LIN {X 0,Y 147.971,Z 1211.135,A -85,B 0,C 180,E1 7432.674,E2 7432.674} C_VEL
LIN {X 0,Y 149.301,Z 1208.656,A -85,B 0,C 180,E1 7429.89,E2 7429.89} C_VEL
LIN {X 0,Y 150.873,Z 1200.807,A -85,B 0,C 180,E1 7422.356,E2 7422.356} C_VEL
LIN {X 0,Y 153.013,Z 1198.113,A -85,B 0,C 180,E1 7420.188,E2 7420.188} C_VEL
LIN {X 0,Y 163,Z 1189.252,A -85,B 0,C 180,E1 7414.094,E2 7414.094} C_VEL
LIN {X 0,Y 174.434,Z 1179.156,A -85,B 0,C 180,E1 7408.716,E2 7408.716} C_VEL
LIN {X 0,Y 189.359,Z 1165.738,A -85,B 0,C 180,E1 7403.252,E2 7403.252} C_VEL
LIN {X 0,Y 205.695,Z 1150.071,A -85,B 0,C 180,E1 7398.578,E2 7398.578} C_VEL
LIN {X 0,Y 219.758,Z 1135.831,A -85,B 0,C 180,E1 7395.296,E2 7395.296} C_VEL
LIN {X 0,Y 236.568,Z 1117.707,A -85,B 0,C 180,E1 7392.022,E2 7392.022} C_VEL
LIN {X 0,Y 253.297,Z 1097.817,A -85,B 0,C 180,E1 7389.298,E2 7389.298} C_VEL
LIN {X 0,Y 266.7,Z 1080.637,A -85,B 0,C 180,E1 7387.42,E2 7387.42} C_VEL
LIN {X 0,Y 282.499,Z 1058.672,A -85,B 0,C 180,E1 7385.484,E2 7385.484} C_VEL
LIN {X 0,Y 297.162,Z 1035.806,A -85,B 0,C 180,E1 7383.912,E2 7383.912} C_VEL
LIN {X 0,Y 309.321,Z 1015.07,A -85,B 0,C 180,E1 7382.764,E2 7382.764} C_VEL
LIN {X 0,Y 323.265,Z 988.553,A -85,B 0,C 180,E1 7381.595,E2 7381.595} C_VEL
LIN {X 0,Y 333.991,Z 965.406,A -85,B 0,C 180,E1 7380.804,E2 7380.804} C_VEL
LIN {X 0,Y 343.958,Z 941.252,A -85,B 0,C 180,E1 7380.142,E2 7380.142} C_VEL
LIN {X 0,Y 353.967,Z 912.892,A -85,B 0,C 180,E1 7379.541,E2 7379.541} C_VEL
LIN {X 0,Y 361.036,Z 888.561,A -85,B 0,C 180,E1 7379.074,E2 7379.074} C_VEL
LIN {X 0,Y 367.735,Z 860.245,A -85,B 0,C 180,E1 7378.576,E2 7378.576} C_VEL
LIN {X 0,Y 376.666,Z 808.206,A -85,B 0,C 180,E1 7377.808,E2 7377.808} C_VEL
LIN {X 0,Y 394.746,Z 699.24,A -85,B 0,C 180,E1 7376.297,E2 7376.297} C_VEL
LIN {X 0,Y 389.783,Z 690.265,A -85,B 0,C 180,E1 7372.557,E2 7372.557} C_VEL
LIN {X 0,Y 385.758,Z 683.234,A -85,B 0,C 180,E1 7369.017,E2 7369.017} C_VEL
LIN {X 0,Y 381.936,Z 676.731,A -85,B 0,C 180,E1 7364.979,E2 7364.979} C_VEL
LIN {X 0,Y 379.584,Z 672.588,A -85,B 0,C 180,E1 7361.975,E2 7361.975} C_VEL
LIN {X 0,Y 378.062,Z 670.252,A -85,B 0,C 180,E1 7359.729,E2 7359.729} C_VEL
LIN {X 0,Y 375.586,Z 667.54,A -85,B 0,C 180,E1 7355.461,E2 7355.461} C_VEL
LIN {X 0,Y 374.446,Z 665.022,A -85,B 0,C 180,E1 7352.112,E2 7352.112} C_VEL
LIN {X 0,Y 373.277,Z 664.346,A -85,B 0,C 180,E1 7346.876,E2 7346.876} C_VEL
LIN {X 0,Y 373.271,Z 664.329,A -85,B 0,C 180,E1 7342.356,E2 7342.356} C_VEL
LIN {X 0,Y 374.579,Z 664.928,A -85,B 0,C 180,E1 7337.311,E2 7337.311} C_VEL
LIN {X 0,Y 375.203,Z 665.478,A -85,B 0,C 180,E1 7335.577,E2 7335.577} C_VEL
LIN {X 0,Y 377.938,Z 669.541,A -85,B 0,C 180,E1 7330.364,E2 7330.364} C_VEL
LIN {X 0,Y 379.465,Z 671.062,A -85,B 0,C 180,E1 7328.258,E2 7328.258} C_VEL
LIN {X 0,Y 383.507,Z 676.422,A -85,B 0,C 180,E1 7323.725,E2 7323.725} C_VEL
LIN {X 0,Y 387.147,Z 681.494,A -85,B 0,C 180,E1 7320.387,E2 7320.387} C_VEL
LIN {X 0,Y 390.659,Z 686.502,A -85,B 0,C 180,E1 7317.598,E2 7317.598} C_VEL
LIN {X 0,Y 391.311,Z 687.552,A -85,B 0,C 180,E1 7317.126,E2 7317.126} C_VEL
LIN {X 0,Y 370.823,Z 810.476,A -85,B 0,C 180,E1 7315.42,E2 7315.42} C_VEL
LIN {X 0,Y 363.996,Z 841.432,A -85,B 0,C 180,E1 7314.831,E2 7314.831} C_VEL
LIN {X 0,Y 357.385,Z 865.622,A -85,B 0,C 180,E1 7314.245,E2 7314.245} C_VEL
LIN {X 0,Y 348.359,Z 893.546,A -85,B 0,C 180,E1 7313.424,E2 7313.424} C_VEL
LIN {X 0,Y 338.511,Z 919.063,A -85,B 0,C 180,E1 7312.498,E2 7312.498} C_VEL
LIN {X 0,Y 328.592,Z 941.804,A -85,B 0,C 180,E1 7311.511,E2 7311.511} C_VEL
LIN {X 0,Y 314.858,Z 969.363,A -85,B 0,C 180,E1 7310.058,E2 7310.058} C_VEL
LIN {X 0,Y 303.618,Z 989.37,A -85,B 0,C 180,E1 7308.778,E2 7308.778} C_VEL
LIN {X 0,Y 290.756,Z 1010.185,A -85,B 0,C 180,E1 7307.202,E2 7307.202} C_VEL
LIN {X 0,Y 274.887,Z 1033.236,A -85,B 0,C 180,E1 7305.056,E2 7305.056} C_VEL
LIN {X 0,Y 261.486,Z 1050.892,A -85,B 0,C 180,E1 7303.039,E2 7303.039} C_VEL
LIN {X 0,Y 247.624,Z 1067.77,A -85,B 0,C 180,E1 7300.704,E2 7300.704} C_VEL
LIN {X 0,Y 229.805,Z 1087.623,A -85,B 0,C 180,E1 7297.233,E2 7297.233} C_VEL
LIN {X 0,Y 215.494,Z 1102.262,A -85,B 0,C 180,E1 7293.968,E2 7293.968} C_VEL
LIN {X 0,Y 201.983,Z 1115.27,A -85,B 0,C 180,E1 7290.344,E2 7290.344} C_VEL
LIN {X 0,Y 185.811,Z 1129.978,A -85,B 0,C 180,E1 7285.061,E2 7285.061} C_VEL
LIN {X 0,Y 172.32,Z 1141.568,A -85,B 0,C 180,E1 7279.48,E2 7279.48} C_VEL
LIN {X 0,Y 161.424,Z 1150.796,A -85,B 0,C 180,E1 7273.761,E2 7273.761} C_VEL
LIN {X 0,Y 151.716,Z 1159.15,A -85,B 0,C 180,E1 7267.118,E2 7267.118} C_VEL
LIN {X 0,Y 142.033,Z 1168.124,A -85,B 0,C 180,E1 7257.649,E2 7257.649} C_VEL
LIN {X 0,Y 136.236,Z 1174.505,A -85,B 0,C 180,E1 7248.471,E2 7248.471} C_VEL
LIN {X 0,Y 133.333,Z 1179.088,A -85,B 0,C 180,E1 7240.102,E2 7240.102} C_VEL
LIN {X 0,Y 132.224,Z 1182.655,A -85,B 0,C 180,E1 7232.12,E2 7232.12} C_VEL
LIN {X 0,Y 132.255,Z 1185.605,A -85,B 0,C 180,E1 7224.096,E2 7224.096} C_VEL
LIN {X 0,Y 133.369,Z 1188.047,A -85,B 0,C 180,E1 7216.105,E2 7216.105} C_VEL
LIN {X 0,Y 136.302,Z 1190.213,A -85,B 0,C 180,E1 7207.164,E2 7207.164} C_VEL
LIN {X 0,Y 142.425,Z 1191.882,A -85,B 0,C 180,E1 7197.586,E2 7197.586} C_VEL
LIN {X 0,Y 153.798,Z 1192.938,A -85,B 0,C 180,E1 7187.208,E2 7187.208} C_VEL
LIN {X 0,Y 173.982,Z 1192.781,A -85,B 0,C 180,E1 7176.278,E2 7176.278} C_VEL
LIN {X 0,Y 180.652,Z 1192.577,A -85,B 0,C 180,E1 7173.594,E2 7173.594} C_VEL
LIN {X 0,Y 156.927,Z 1204.45,A -85,B 0,C 180,E1 7162.792,E2 7162.792} C_VEL
LIN {X 0,Y 144.33,Z 1211.835,A -85,B 0,C 180,E1 7153.302,E2 7153.302} C_VEL
LIN {X 0,Y 136.328,Z 1217.665,A -85,B 0,C 180,E1 7143.266,E2 7143.266} C_VEL
LIN {X 0,Y 132.398,Z 1221.841,A -85,B 0,C 180,E1 7133.594,E2 7133.594} C_VEL
LIN {X 0,Y 131.351,Z 1224.76,A -85,B 0,C 180,E1 7124.098,E2 7124.098} C_VEL
LIN {X 0,Y 132.003,Z 1226.283,A -85,B 0,C 180,E1 7116.087,E2 7116.087} C_VEL
LIN {X 0,Y 132.577,Z 1226.521,A -85,B 0,C 180,E1 7110.864,E2 7110.864} C_VEL
LIN {X 0,Y 132.4,Z 1226.185,A -85,B 0,C 180,E1 7106.103,E2 7106.103} C_VEL
LIN {X 0,Y 131.668,Z 1224.515,A -85,B 0,C 180,E1 7098.415,E2 7098.415} C_VEL
LIN {X 0,Y 132.136,Z 1221.245,A -85,B 0,C 180,E1 7089.63,E2 7089.63} C_VEL
LIN {X 0,Y 134.667,Z 1216.788,A -85,B 0,C 180,E1 7081.144,E2 7081.144} C_VEL
LIN {X 0,Y 139.462,Z 1211.063,A -85,B 0,C 180,E1 7072.969,E2 7072.969} C_VEL
LIN {X 0,Y 146.512,Z 1204.062,A -85,B 0,C 180,E1 7065.338,E2 7065.338} C_VEL
LIN {X 0,Y 153.013,Z 1198.113,A -85,B 0,C 180,E1 7060.188,E2 7060.188} C_VEL
LIN {X 0,Y 155.592,Z 1194.978,A -85,B 0,C 180,E1 7057.733,E2 7057.733} C_VEL
LIN {X 0,Y 160.318,Z 1185.779,A -85,B 0,C 180,E1 7050.981,E2 7050.981} C_VEL
LIN {X 0,Y 163.262,Z 1182.63,A -85,B 0,C 180,E1 7049.177,E2 7049.177} C_VEL
LIN {X 0,Y 177.711,Z 1170.122,A -85,B 0,C 180,E1 7043.494,E2 7043.494} C_VEL
LIN {X 0,Y 190.823,Z 1158.366,A -85,B 0,C 180,E1 7039.41,E2 7039.41} C_VEL
LIN {X 0,Y 205.591,Z 1144.445,A -85,B 0,C 180,E1 7035.644,E2 7035.644} C_VEL
LIN {X 0,Y 223.87,Z 1125.852,A -85,B 0,C 180,E1 7031.856,E2 7031.856} C_VEL
LIN {X 0,Y 238.619,Z 1109.591,A -85,B 0,C 180,E1 7029.318,E2 7029.318} C_VEL
LIN {X 0,Y 253.429,Z 1092.024,A -85,B 0,C 180,E1 7027.13,E2 7027.13} C_VEL
LIN {X 0,Y 270.961,Z 1069.146,A -85,B 0,C 180,E1 7024.911,E2 7024.911} C_VEL
LIN {X 0,Y 284.524,Z 1049.638,A -85,B 0,C 180,E1 7023.425,E2 7023.425} C_VEL
LIN {X 0,Y 298.655,Z 1027.411,A -85,B 0,C 180,E1 7022.055,E2 7022.055} C_VEL
LIN {X 0,Y 312.994,Z 1002.012,A -85,B 0,C 180,E1 7020.833,E2 7020.833} C_VEL
LIN {X 0,Y 324.089,Z 980.101,A -85,B 0,C 180,E1 7020,E2 7020} C_VEL
LIN {X 0,Y 336.152,Z 953.318,A -85,B 0,C 180,E1 7019.194,E2 7019.194} C_VEL
LIN {X 0,Y 346.059,Z 927.667,A -85,B 0,C 180,E1 7018.611,E2 7018.611} C_VEL
LIN {X 0,Y 353.888,Z 904.184,A -85,B 0,C 180,E1 7018.161,E2 7018.161} C_VEL
LIN {X 0,Y 362.217,Z 873.201,A -85,B 0,C 180,E1 7017.606,E2 7017.606} C_VEL
LIN {X 0,Y 367.389,Z 848.457,A -85,B 0,C 180,E1 7017.212,E2 7017.212} C_VEL
LIN {X 0,Y 391.677,Z 704.829,A -85,B 0,C 180,E1 7015.241,E2 7015.241} C_VEL
LIN {X 0,Y 387.34,Z 696.911,A -85,B 0,C 180,E1 7011.838,E2 7011.838} C_VEL
LIN {X 0,Y 383.448,Z 689.926,A -85,B 0,C 180,E1 7008.264,E2 7008.264} C_VEL
LIN {X 0,Y 379.941,Z 683.925,A -85,B 0,C 180,E1 7004.405,E2 7004.405} C_VEL
LIN {X 0,Y 377.891,Z 680.307,A -85,B 0,C 180,E1 7001.785,E2 7001.785} C_VEL
LIN {X 0,Y 376.435,Z 678.064,A -85,B 0,C 180,E1 6999.637,E2 6999.637} C_VEL
LIN {X 0,Y 373.974,Z 675.341,A -85,B 0,C 180,E1 6995.348,E2 6995.348} C_VEL
LIN {X 0,Y 372.85,Z 672.853,A -85,B 0,C 180,E1 6992.011,E2 6992.011} C_VEL
LIN {X 0,Y 371.661,Z 672.174,A -85,B 0,C 180,E1 6986.529,E2 6986.529} C_VEL
LIN {X 0,Y 371.769,Z 672.176,A -85,B 0,C 180,E1 6981.982,E2 6981.982} C_VEL
LIN {X 0,Y 373.313,Z 672.915,A -85,B 0,C 180,E1 6976.5,E2 6976.5} C_VEL
LIN {X 0,Y 373.744,Z 673.675,A -85,B 0,C 180,E1 6975.282,E2 6975.282} C_VEL
